   1:  PR[GP1:91,1] = PR[GP1:90,1] + -5.573;
   1:  PR[GP1:91,2] = PR[GP1:90,2] + 6.537;
   1:L PR[91] R[100]mm/sec CNT100;
   1:  PR[GP1:91,1] = PR[GP1:90,1] + -6.753;
   1:  PR[GP1:91,2] = PR[GP1:90,2] + 9.038;
   1:L PR[91] R[100]mm/sec CNT100;
   1:  PR[GP1:91,1] = PR[GP1:90,1] + -7.010;
   1:  PR[GP1:91,2] = PR[GP1:90,2] + 9.357;
   1:L PR[91] R[100]mm/sec CNT100;
   1:  PR[GP1:91,1] = PR[GP1:90,1] + -8.709;
   1:  PR[GP1:91,2] = PR[GP1:90,2] + 11.817;
   1:L PR[91] R[100]mm/sec CNT100;
   1:  PR[GP1:91,1] = PR[GP1:90,1] + -10.629;
   1:  PR[GP1:91,2] = PR[GP1:90,2] + 13.805;
   1:L PR[91] R[100]mm/sec CNT100;
   1:  PR[GP1:91,1] = PR[GP1:90,1] + -10.976;
   1:  PR[GP1:91,2] = PR[GP1:90,2] + 14.025;
   1:L PR[91] R[100]mm/sec CNT100;
   1:  PR[GP1:91,1] = PR[GP1:90,1] + -13.376;
   1:  PR[GP1:91,2] = PR[GP1:90,2] + 15.808;
   1:L PR[91] R[100]mm/sec CNT100;
   1:  PR[GP1:91,1] = PR[GP1:90,1] + -15.833;
   1:  PR[GP1:91,2] = PR[GP1:90,2] + 17.073;
   1:L PR[91] R[100]mm/sec CNT100;
   1:  PR[GP1:91,1] = PR[GP1:90,1] + -16.233;
   1:  PR[GP1:91,2] = PR[GP1:90,2] + 17.169;
   1:L PR[91] R[100]mm/sec CNT100;
   1:  PR[GP1:91,1] = PR[GP1:90,1] + -19.079;
   1:  PR[GP1:91,2] = PR[GP1:90,2] + 18.086;
   1:L PR[91] R[100]mm/sec CNT100;
   1:  PR[GP1:91,1] = PR[GP1:90,1] + -21.812;
   1:  PR[GP1:91,2] = PR[GP1:90,2] + 18.493;
   1:L PR[91] R[100]mm/sec CNT100;
   1:  PR[GP1:91,1] = PR[GP1:90,1] + -22.221;
   1:  PR[GP1:91,2] = PR[GP1:90,2] + 18.455;
   1:L PR[91] R[100]mm/sec CNT100;
   1:  PR[GP1:91,1] = PR[GP1:90,1] + -25.212;
   1:  PR[GP1:91,2] = PR[GP1:90,2] + 18.408;
   1:L PR[91] R[100]mm/sec CNT100;
   1:  PR[GP1:91,1] = PR[GP1:90,1] + -27.929;
   1:  PR[GP1:91,2] = PR[GP1:90,2] + 17.915;
   1:L PR[91] R[100]mm/sec CNT100;
   1:  PR[GP1:91,1] = PR[GP1:90,1] + -28.304;
   1:  PR[GP1:91,2] = PR[GP1:90,2] + 17.747;
   1:L PR[91] R[100]mm/sec CNT100;
   1:  PR[GP1:91,1] = PR[GP1:90,1] + -31.122;
   1:  PR[GP1:91,2] = PR[GP1:90,2] + 16.741;
   1:L PR[91] R[100]mm/sec CNT100;
   1:  PR[GP1:91,1] = PR[GP1:90,1] + -33.536;
   1:  PR[GP1:91,2] = PR[GP1:90,2] + 15.401;
   1:L PR[91] R[100]mm/sec CNT100;
   1:  PR[GP1:91,1] = PR[GP1:90,1] + -33.837;
   1:  PR[GP1:91,2] = PR[GP1:90,2] + 15.121;
   1:L PR[91] R[100]mm/sec CNT100;
   1:  PR[GP1:91,1] = PR[GP1:90,1] + -36.182;
   1:  PR[GP1:91,2] = PR[GP1:90,2] + 13.261;
   1:L PR[91] R[100]mm/sec CNT100;
   1:  PR[GP1:91,1] = PR[GP1:90,1] + -38.036;
   1:  PR[GP1:91,2] = PR[GP1:90,2] + 11.216;
   1:L PR[91] R[100]mm/sec CNT100;
   1:  PR[GP1:91,1] = PR[GP1:90,1] + -38.230;
   1:  PR[GP1:91,2] = PR[GP1:90,2] + 10.854;
   1:L PR[91] R[100]mm/sec CNT100;
   1:  PR[GP1:91,1] = PR[GP1:90,1] + -39.853;
   1:  PR[GP1:91,2] = PR[GP1:90,2] + 8.338;
   1:L PR[91] R[100]mm/sec CNT100;
   1:  PR[GP1:91,1] = PR[GP1:90,1] + -40.951;
   1:  PR[GP1:91,2] = PR[GP1:90,2] + 5.807;
   1:L PR[91] R[100]mm/sec CNT100;
   1:  PR[GP1:91,1] = PR[GP1:90,1] + -41.018;
   1:  PR[GP1:91,2] = PR[GP1:90,2] + 5.402;
   1:L PR[91] R[100]mm/sec CNT100;
   1:  PR[GP1:91,1] = PR[GP1:90,1] + -41.746;
   1:  PR[GP1:91,2] = PR[GP1:90,2] + 2.497;
   1:L PR[91] R[100]mm/sec CNT100;
   1:  PR[GP1:91,1] = PR[GP1:90,1] + -41.972;
   1:  PR[GP1:91,2] = PR[GP1:90,2] + -0.252;
   1:L PR[91] R[100]mm/sec CNT100;
   1:  PR[GP1:91,1] = PR[GP1:90,1] + -41.905;
   1:  PR[GP1:91,2] = PR[GP1:90,2] + -0.657;
   1:L PR[91] R[100]mm/sec CNT100;
   1:  PR[GP1:91,1] = PR[GP1:90,1] + -41.660;
   1:  PR[GP1:91,2] = PR[GP1:90,2] + -3.643;
   1:L PR[91] R[100]mm/sec CNT100;
   1:  PR[GP1:91,1] = PR[GP1:90,1] + -40.975;
   1:  PR[GP1:91,2] = PR[GP1:90,2] + -6.377;
   1:L PR[91] R[100]mm/sec CNT100;
   1:  PR[GP1:91,1] = PR[GP1:90,1] + -39.830;
   1:  PR[GP1:91,2] = PR[GP1:90,2] + -9.016;
   1:L PR[91] R[100]mm/sec CNT100;
   1:  PR[GP1:91,1] = PR[GP1:90,1] + -39.636;
   1:  PR[GP1:91,2] = PR[GP1:90,2] + -9.378;
   1:L PR[91] R[100]mm/sec CNT100;
   1:  PR[GP1:91,1] = PR[GP1:90,1] + -38.075;
   1:  PR[GP1:91,2] = PR[GP1:90,2] + -11.797;
   1:L PR[91] R[100]mm/sec CNT100;
   1:  PR[GP1:91,1] = PR[GP1:90,1] + -36.144;
   1:  PR[GP1:91,2] = PR[GP1:90,2] + -13.927;
   1:L PR[91] R[100]mm/sec CNT100;
   1:  PR[GP1:91,1] = PR[GP1:90,1] + -35.842;
   1:  PR[GP1:91,2] = PR[GP1:90,2] + -14.207;
   1:L PR[91] R[100]mm/sec CNT100;
   1:  PR[GP1:91,1] = PR[GP1:90,1] + -33.586;
   1:  PR[GP1:91,2] = PR[GP1:90,2] + -15.997;
   1:L PR[91] R[100]mm/sec CNT100;
   1:  PR[GP1:91,1] = PR[GP1:90,1] + -31.073;
   1:  PR[GP1:91,2] = PR[GP1:90,2] + -17.392;
   1:L PR[91] R[100]mm/sec CNT100;
   1:  PR[GP1:91,1] = PR[GP1:90,1] + -30.697;
   1:  PR[GP1:91,2] = PR[GP1:90,2] + -17.560;
   1:L PR[91] R[100]mm/sec CNT100;
   1:  PR[GP1:91,1] = PR[GP1:90,1] + -27.985;
   1:  PR[GP1:91,2] = PR[GP1:90,2] + -18.529;
   1:L PR[91] R[100]mm/sec CNT100;
   1:  PR[GP1:91,1] = PR[GP1:90,1] + -25.157;
   1:  PR[GP1:91,2] = PR[GP1:90,2] + -19.042;
   1:L PR[91] R[100]mm/sec CNT100;
   1:  PR[GP1:91,1] = PR[GP1:90,1] + -24.748;
   1:  PR[GP1:91,2] = PR[GP1:90,2] + -19.080;
   1:L PR[91] R[100]mm/sec CNT100;
   1:  PR[GP1:91,1] = PR[GP1:90,1] + -21.867;
   1:  PR[GP1:91,2] = PR[GP1:90,2] + -19.125;
   1:L PR[91] R[100]mm/sec CNT100;
   1:  PR[GP1:91,1] = PR[GP1:90,1] + -19.025;
   1:  PR[GP1:91,2] = PR[GP1:90,2] + -18.702;
   1:L PR[91] R[100]mm/sec CNT100;
   1:  PR[GP1:91,1] = PR[GP1:90,1] + -18.625;
   1:  PR[GP1:91,2] = PR[GP1:90,2] + -18.606;
   1:L PR[91] R[100]mm/sec CNT100;
   1:  PR[GP1:91,1] = PR[GP1:90,1] + -15.882;
   1:  PR[GP1:91,2] = PR[GP1:90,2] + -17.722;
   1:L PR[91] R[100]mm/sec CNT100;
   1:  PR[GP1:91,1] = PR[GP1:90,1] + -13.329;
   1:  PR[GP1:91,2] = PR[GP1:90,2] + -16.408;
   1:L PR[91] R[100]mm/sec CNT100;
   1:  PR[GP1:91,1] = PR[GP1:90,1] + -12.981;
   1:  PR[GP1:91,2] = PR[GP1:90,2] + -16.187;
   1:L PR[91] R[100]mm/sec CNT100;
   1:  PR[GP1:91,1] = PR[GP1:90,1] + -10.667;
   1:  PR[GP1:91,2] = PR[GP1:90,2] + -14.468;
   1:L PR[91] R[100]mm/sec CNT100;
   1:  PR[GP1:91,1] = PR[GP1:90,1] + -8.672;
   1:  PR[GP1:91,2] = PR[GP1:90,2] + -12.403;
   1:L PR[91] R[100]mm/sec CNT100;
   1:  PR[GP1:91,1] = PR[GP1:90,1] + -8.414;
   1:  PR[GP1:91,2] = PR[GP1:90,2] + -12.082;
   1:L PR[91] R[100]mm/sec CNT100;
   1:  PR[GP1:91,1] = PR[GP1:90,1] + -6.775;
   1:  PR[GP1:91,2] = PR[GP1:90,2] + -9.710;
   1:L PR[91] R[100]mm/sec CNT100;
   1:  PR[GP1:91,1] = PR[GP1:90,1] + -5.551;
   1:  PR[GP1:91,2] = PR[GP1:90,2] + -7.113;
   1:L PR[91] R[100]mm/sec CNT100;
   1:  PR[GP1:91,1] = PR[GP1:90,1] + -5.411;
   1:  PR[GP1:91,2] = PR[GP1:90,2] + -6.729;
   1:L PR[91] R[100]mm/sec CNT100;
   1:  PR[GP1:91,1] = PR[GP1:90,1] + -4.557;
   1:  PR[GP1:91,2] = PR[GP1:90,2] + -3.704;
   1:L PR[91] R[100]mm/sec CNT100;
   1:  PR[GP1:91,1] = PR[GP1:90,1] + -4.234;
   1:  PR[GP1:91,2] = PR[GP1:90,2] + -2.880;
   1:L PR[91] R[100]mm/sec CNT100;
   1:  PR[GP1:91,1] = PR[GP1:90,1] + -3.519;
   1:  PR[GP1:91,2] = PR[GP1:90,2] + -2.050;
   1:L PR[91] R[100]mm/sec CNT100;
   1:  PR[GP1:91,1] = PR[GP1:90,1] + -2.563;
   1:  PR[GP1:91,2] = PR[GP1:90,2] + -1.510;
   1:L PR[91] R[100]mm/sec CNT100;
   1:  PR[GP1:91,1] = PR[GP1:90,1] + -2.182;
   1:  PR[GP1:91,2] = PR[GP1:90,2] + -1.443;
   1:L PR[91] R[100]mm/sec CNT100;
   1:  PR[GP1:91,1] = PR[GP1:90,1] + -1.745;
   1:  PR[GP1:91,2] = PR[GP1:90,2] + -1.269;
   1:L PR[91] R[100]mm/sec CNT100;
   1:  PR[GP1:91,1] = PR[GP1:90,1] + 1.895;
   1:  PR[GP1:91,2] = PR[GP1:90,2] + -1.275;
   1:L PR[91] R[100]mm/sec CNT100;
   1:  PR[GP1:91,1] = PR[GP1:90,1] + 2.330;
   1:  PR[GP1:91,2] = PR[GP1:90,2] + -1.442;
   1:L PR[91] R[100]mm/sec CNT100;
   1:  PR[GP1:91,1] = PR[GP1:90,1] + 2.720;
   1:  PR[GP1:91,2] = PR[GP1:90,2] + -1.510;
   1:L PR[91] R[100]mm/sec CNT100;
   1:  PR[GP1:91,1] = PR[GP1:90,1] + 3.676;
   1:  PR[GP1:91,2] = PR[GP1:90,2] + -2.050;
   1:L PR[91] R[100]mm/sec CNT100;
   1:  PR[GP1:91,1] = PR[GP1:90,1] + 4.391;
   1:  PR[GP1:91,2] = PR[GP1:90,2] + -2.881;
   1:L PR[91] R[100]mm/sec CNT100;
   1:  PR[GP1:91,1] = PR[GP1:90,1] + 4.700;
   1:  PR[GP1:91,2] = PR[GP1:90,2] + -3.670;
   1:L PR[91] R[100]mm/sec CNT100;
   1:  PR[GP1:91,1] = PR[GP1:90,1] + 4.916;
   1:  PR[GP1:91,2] = PR[GP1:90,2] + -4.299;
   1:L PR[91] R[100]mm/sec CNT100;
   1:  PR[GP1:91,1] = PR[GP1:90,1] + 5.730;
   1:  PR[GP1:91,2] = PR[GP1:90,2] + -7.161;
   1:L PR[91] R[100]mm/sec CNT100;
   1:  PR[GP1:91,1] = PR[GP1:90,1] + 6.909;
   1:  PR[GP1:91,2] = PR[GP1:90,2] + -9.661;
   1:L PR[91] R[100]mm/sec CNT100;
   1:  PR[GP1:91,1] = PR[GP1:90,1] + 7.167;
   1:  PR[GP1:91,2] = PR[GP1:90,2] + -9.981;
   1:L PR[91] R[100]mm/sec CNT100;
   1:  PR[GP1:91,1] = PR[GP1:90,1] + 8.866;
   1:  PR[GP1:91,2] = PR[GP1:90,2] + -12.441;
   1:L PR[91] R[100]mm/sec CNT100;
   1:  PR[GP1:91,1] = PR[GP1:90,1] + 10.786;
   1:  PR[GP1:91,2] = PR[GP1:90,2] + -14.429;
   1:L PR[91] R[100]mm/sec CNT100;
   1:  PR[GP1:91,1] = PR[GP1:90,1] + 11.133;
   1:  PR[GP1:91,2] = PR[GP1:90,2] + -14.649;
   1:L PR[91] R[100]mm/sec CNT100;
   1:  PR[GP1:91,1] = PR[GP1:90,1] + 13.533;
   1:  PR[GP1:91,2] = PR[GP1:90,2] + -16.432;
   1:L PR[91] R[100]mm/sec CNT100;
   1:  PR[GP1:91,1] = PR[GP1:90,1] + 15.990;
   1:  PR[GP1:91,2] = PR[GP1:90,2] + -17.697;
   1:L PR[91] R[100]mm/sec CNT100;
   1:  PR[GP1:91,1] = PR[GP1:90,1] + 16.389;
   1:  PR[GP1:91,2] = PR[GP1:90,2] + -17.793;
   1:L PR[91] R[100]mm/sec CNT100;
   1:  PR[GP1:91,1] = PR[GP1:90,1] + 19.236;
   1:  PR[GP1:91,2] = PR[GP1:90,2] + -18.710;
   1:L PR[91] R[100]mm/sec CNT100;
   1:  PR[GP1:91,1] = PR[GP1:90,1] + 21.968;
   1:  PR[GP1:91,2] = PR[GP1:90,2] + -19.117;
   1:L PR[91] R[100]mm/sec CNT100;
   1:  PR[GP1:91,1] = PR[GP1:90,1] + 22.377;
   1:  PR[GP1:91,2] = PR[GP1:90,2] + -19.079;
   1:L PR[91] R[100]mm/sec CNT100;
   1:  PR[GP1:91,1] = PR[GP1:90,1] + 25.369;
   1:  PR[GP1:91,2] = PR[GP1:90,2] + -19.032;
   1:L PR[91] R[100]mm/sec CNT100;
   1:  PR[GP1:91,1] = PR[GP1:90,1] + 28.086;
   1:  PR[GP1:91,2] = PR[GP1:90,2] + -18.539;
   1:L PR[91] R[100]mm/sec CNT100;
   1:  PR[GP1:91,1] = PR[GP1:90,1] + 28.461;
   1:  PR[GP1:91,2] = PR[GP1:90,2] + -18.371;
   1:L PR[91] R[100]mm/sec CNT100;
   1:  PR[GP1:91,1] = PR[GP1:90,1] + 31.279;
   1:  PR[GP1:91,2] = PR[GP1:90,2] + -17.365;
   1:L PR[91] R[100]mm/sec CNT100;
   1:  PR[GP1:91,1] = PR[GP1:90,1] + 33.693;
   1:  PR[GP1:91,2] = PR[GP1:90,2] + -16.025;
   1:L PR[91] R[100]mm/sec CNT100;
   1:  PR[GP1:91,1] = PR[GP1:90,1] + 33.993;
   1:  PR[GP1:91,2] = PR[GP1:90,2] + -15.745;
   1:L PR[91] R[100]mm/sec CNT100;
   1:  PR[GP1:91,1] = PR[GP1:90,1] + 36.339;
   1:  PR[GP1:91,2] = PR[GP1:90,2] + -13.885;
   1:L PR[91] R[100]mm/sec CNT100;
   1:  PR[GP1:91,1] = PR[GP1:90,1] + 38.193;
   1:  PR[GP1:91,2] = PR[GP1:90,2] + -11.840;
   1:L PR[91] R[100]mm/sec CNT100;
   1:  PR[GP1:91,1] = PR[GP1:90,1] + 38.387;
   1:  PR[GP1:91,2] = PR[GP1:90,2] + -11.478;
   1:L PR[91] R[100]mm/sec CNT100;
   1:  PR[GP1:91,1] = PR[GP1:90,1] + 40.010;
   1:  PR[GP1:91,2] = PR[GP1:90,2] + -8.962;
   1:L PR[91] R[100]mm/sec CNT100;
   1:  PR[GP1:91,1] = PR[GP1:90,1] + 41.108;
   1:  PR[GP1:91,2] = PR[GP1:90,2] + -6.431;
   1:L PR[91] R[100]mm/sec CNT100;
   1:  PR[GP1:91,1] = PR[GP1:90,1] + 41.175;
   1:  PR[GP1:91,2] = PR[GP1:90,2] + -6.026;
   1:L PR[91] R[100]mm/sec CNT100;
   1:  PR[GP1:91,1] = PR[GP1:90,1] + 41.903;
   1:  PR[GP1:91,2] = PR[GP1:90,2] + -3.121;
   1:L PR[91] R[100]mm/sec CNT100;
   1:  PR[GP1:91,1] = PR[GP1:90,1] + 42.129;
   1:  PR[GP1:91,2] = PR[GP1:90,2] + -0.372;
   1:L PR[91] R[100]mm/sec CNT100;
   1:  PR[GP1:91,1] = PR[GP1:90,1] + 42.061;
   1:  PR[GP1:91,2] = PR[GP1:90,2] + 0.033;
   1:L PR[91] R[100]mm/sec CNT100;
   1:  PR[GP1:91,1] = PR[GP1:90,1] + 41.817;
   1:  PR[GP1:91,2] = PR[GP1:90,2] + 3.019;
   1:L PR[91] R[100]mm/sec CNT100;
   1:  PR[GP1:91,1] = PR[GP1:90,1] + 41.132;
   1:  PR[GP1:91,2] = PR[GP1:90,2] + 5.753;
   1:L PR[91] R[100]mm/sec CNT100;
   1:  PR[GP1:91,1] = PR[GP1:90,1] + 39.987;
   1:  PR[GP1:91,2] = PR[GP1:90,2] + 8.392;
   1:L PR[91] R[100]mm/sec CNT100;
   1:  PR[GP1:91,1] = PR[GP1:90,1] + 39.792;
   1:  PR[GP1:91,2] = PR[GP1:90,2] + 8.754;
   1:L PR[91] R[100]mm/sec CNT100;
   1:  PR[GP1:91,1] = PR[GP1:90,1] + 38.232;
   1:  PR[GP1:91,2] = PR[GP1:90,2] + 11.173;
   1:L PR[91] R[100]mm/sec CNT100;
   1:  PR[GP1:91,1] = PR[GP1:90,1] + 36.300;
   1:  PR[GP1:91,2] = PR[GP1:90,2] + 13.303;
   1:L PR[91] R[100]mm/sec CNT100;
   1:  PR[GP1:91,1] = PR[GP1:90,1] + 35.999;
   1:  PR[GP1:91,2] = PR[GP1:90,2] + 13.583;
   1:L PR[91] R[100]mm/sec CNT100;
   1:  PR[GP1:91,1] = PR[GP1:90,1] + 33.743;
   1:  PR[GP1:91,2] = PR[GP1:90,2] + 15.373;
   1:L PR[91] R[100]mm/sec CNT100;
   1:  PR[GP1:91,1] = PR[GP1:90,1] + 31.230;
   1:  PR[GP1:91,2] = PR[GP1:90,2] + 16.768;
   1:L PR[91] R[100]mm/sec CNT100;
   1:  PR[GP1:91,1] = PR[GP1:90,1] + 30.854;
   1:  PR[GP1:91,2] = PR[GP1:90,2] + 16.936;
   1:L PR[91] R[100]mm/sec CNT100;
   1:  PR[GP1:91,1] = PR[GP1:90,1] + 28.142;
   1:  PR[GP1:91,2] = PR[GP1:90,2] + 17.905;
   1:L PR[91] R[100]mm/sec CNT100;
   1:  PR[GP1:91,1] = PR[GP1:90,1] + 25.314;
   1:  PR[GP1:91,2] = PR[GP1:90,2] + 18.418;
   1:L PR[91] R[100]mm/sec CNT100;
   1:  PR[GP1:91,1] = PR[GP1:90,1] + 24.904;
   1:  PR[GP1:91,2] = PR[GP1:90,2] + 18.456;
   1:L PR[91] R[100]mm/sec CNT100;
   1:  PR[GP1:91,1] = PR[GP1:90,1] + 22.024;
   1:  PR[GP1:91,2] = PR[GP1:90,2] + 18.501;
   1:L PR[91] R[100]mm/sec CNT100;
   1:  PR[GP1:91,1] = PR[GP1:90,1] + 19.182;
   1:  PR[GP1:91,2] = PR[GP1:90,2] + 18.078;
   1:L PR[91] R[100]mm/sec CNT100;
   1:  PR[GP1:91,1] = PR[GP1:90,1] + 18.782;
   1:  PR[GP1:91,2] = PR[GP1:90,2] + 17.982;
   1:L PR[91] R[100]mm/sec CNT100;
   1:  PR[GP1:91,1] = PR[GP1:90,1] + 16.039;
   1:  PR[GP1:91,2] = PR[GP1:90,2] + 17.098;
   1:L PR[91] R[100]mm/sec CNT100;
   1:  PR[GP1:91,1] = PR[GP1:90,1] + 13.485;
   1:  PR[GP1:91,2] = PR[GP1:90,2] + 15.784;
   1:L PR[91] R[100]mm/sec CNT100;
   1:  PR[GP1:91,1] = PR[GP1:90,1] + 13.138;
   1:  PR[GP1:91,2] = PR[GP1:90,2] + 15.563;
   1:L PR[91] R[100]mm/sec CNT100;
   1:  PR[GP1:91,1] = PR[GP1:90,1] + 10.824;
   1:  PR[GP1:91,2] = PR[GP1:90,2] + 13.844;
   1:L PR[91] R[100]mm/sec CNT100;
   1:  PR[GP1:91,1] = PR[GP1:90,1] + 8.829;
   1:  PR[GP1:91,2] = PR[GP1:90,2] + 11.779;
   1:L PR[91] R[100]mm/sec CNT100;
   1:  PR[GP1:91,1] = PR[GP1:90,1] + 8.571;
   1:  PR[GP1:91,2] = PR[GP1:90,2] + 11.459;
   1:L PR[91] R[100]mm/sec CNT100;
   1:  PR[GP1:91,1] = PR[GP1:90,1] + 6.932;
   1:  PR[GP1:91,2] = PR[GP1:90,2] + 9.086;
   1:L PR[91] R[100]mm/sec CNT100;
   1:  PR[GP1:91,1] = PR[GP1:90,1] + 5.708;
   1:  PR[GP1:91,2] = PR[GP1:90,2] + 6.489;
   1:L PR[91] R[100]mm/sec CNT100;
   1:  PR[GP1:91,1] = PR[GP1:90,1] + 5.568;
   1:  PR[GP1:91,2] = PR[GP1:90,2] + 6.105;
   1:L PR[91] R[100]mm/sec CNT100;
   1:  PR[GP1:91,1] = PR[GP1:90,1] + 4.714;
   1:  PR[GP1:91,2] = PR[GP1:90,2] + 3.080;
   1:L PR[91] R[100]mm/sec CNT100;
   1:  PR[GP1:91,1] = PR[GP1:90,1] + 4.391;
   1:  PR[GP1:91,2] = PR[GP1:90,2] + 2.256;
   1:L PR[91] R[100]mm/sec CNT100;
   1:  PR[GP1:91,1] = PR[GP1:90,1] + 3.676;
   1:  PR[GP1:91,2] = PR[GP1:90,2] + 1.426;
   1:L PR[91] R[100]mm/sec CNT100;
   1:  PR[GP1:91,1] = PR[GP1:90,1] + 2.720;
   1:  PR[GP1:91,2] = PR[GP1:90,2] + 0.886;
   1:L PR[91] R[100]mm/sec CNT100;
   1:  PR[GP1:91,1] = PR[GP1:90,1] + 2.341;
   1:  PR[GP1:91,2] = PR[GP1:90,2] + 0.820;
   1:L PR[91] R[100]mm/sec CNT100;
   1:  PR[GP1:91,1] = PR[GP1:90,1] + 1.903;
   1:  PR[GP1:91,2] = PR[GP1:90,2] + 0.644;
   1:L PR[91] R[100]mm/sec CNT100;
   1:  PR[GP1:91,1] = PR[GP1:90,1] + -1.738;
   1:  PR[GP1:91,2] = PR[GP1:90,2] + 0.651;
   1:L PR[91] R[100]mm/sec CNT100;
   1:  PR[91] = PR[90];
   1:  PR[GP1:91,1] = PR[GP1:90,1] + -2.253;
   1:  PR[GP1:91,2] = PR[GP1:90,2] + 0.908;
   1:  PR[GP1:91,3] = PR[GP1:90,3] + 5.185;
   1:L PR[91] R[100]mm/sec CNT100;
   1:  PR[GP1:91,1] = PR[GP1:90,1] + -2.647;
   1:  PR[GP1:91,2] = PR[GP1:90,2] + 1.025;
   1:L PR[91] R[100]mm/sec CNT100;
   1:  PR[GP1:91,1] = PR[GP1:90,1] + -3.536;
   1:  PR[GP1:91,2] = PR[GP1:90,2] + 1.523;
   1:L PR[91] R[100]mm/sec CNT100;
   1:  PR[GP1:91,1] = PR[GP1:90,1] + -4.259;
   1:  PR[GP1:91,2] = PR[GP1:90,2] + 2.372;
   1:L PR[91] R[100]mm/sec CNT100;
   1:  PR[GP1:91,1] = PR[GP1:90,1] + -4.588;
   1:  PR[GP1:91,2] = PR[GP1:90,2] + 3.246;
   1:L PR[91] R[100]mm/sec CNT100;
   1:  PR[GP1:91,1] = PR[GP1:90,1] + -5.418;
   1:  PR[GP1:91,2] = PR[GP1:90,2] + 6.210;
   1:L PR[91] R[100]mm/sec CNT100;
   1:  PR[GP1:91,1] = PR[GP1:90,1] + -6.705;
   1:  PR[GP1:91,2] = PR[GP1:90,2] + 8.939;
   1:L PR[91] R[100]mm/sec CNT100;
   1:  PR[GP1:91,1] = PR[GP1:90,1] + -6.791;
   1:  PR[GP1:91,2] = PR[GP1:90,2] + 9.139;
   1:L PR[91] R[100]mm/sec CNT100;
   1:  PR[GP1:91,1] = PR[GP1:90,1] + -8.462;
   1:  PR[GP1:91,2] = PR[GP1:90,2] + 11.559;
   1:L PR[91] R[100]mm/sec CNT100;
   1:  PR[GP1:91,1] = PR[GP1:90,1] + -8.569;
   1:  PR[GP1:91,2] = PR[GP1:90,2] + 11.694;
   1:L PR[91] R[100]mm/sec CNT100;
   1:  PR[GP1:91,1] = PR[GP1:90,1] + -10.621;
   1:  PR[GP1:91,2] = PR[GP1:90,2] + 13.818;
   1:L PR[91] R[100]mm/sec CNT100;
   1:  PR[GP1:91,1] = PR[GP1:90,1] + -13.178;
   1:  PR[GP1:91,2] = PR[GP1:90,2] + 15.718;
   1:L PR[91] R[100]mm/sec CNT100;
   1:  PR[GP1:91,1] = PR[GP1:90,1] + -15.815;
   1:  PR[GP1:91,2] = PR[GP1:90,2] + 17.075;
   1:L PR[91] R[100]mm/sec CNT100;
   1:  PR[GP1:91,1] = PR[GP1:90,1] + -15.944;
   1:  PR[GP1:91,2] = PR[GP1:90,2] + 17.127;
   1:L PR[91] R[100]mm/sec CNT100;
   1:  PR[GP1:91,1] = PR[GP1:90,1] + -18.795;
   1:  PR[GP1:91,2] = PR[GP1:90,2] + 18.045;
   1:L PR[91] R[100]mm/sec CNT100;
   1:  PR[GP1:91,1] = PR[GP1:90,1] + -21.788;
   1:  PR[GP1:91,2] = PR[GP1:90,2] + 18.491;
   1:L PR[91] R[100]mm/sec CNT100;
   1:  PR[GP1:91,1] = PR[GP1:90,1] + -21.912;
   1:  PR[GP1:91,2] = PR[GP1:90,2] + 18.506;
   1:L PR[91] R[100]mm/sec CNT100;
   1:  PR[GP1:91,1] = PR[GP1:90,1] + -24.871;
   1:  PR[GP1:91,2] = PR[GP1:90,2] + 18.460;
   1:L PR[91] R[100]mm/sec CNT100;
   1:  PR[GP1:91,1] = PR[GP1:90,1] + -27.991;
   1:  PR[GP1:91,2] = PR[GP1:90,2] + 17.902;
   1:L PR[91] R[100]mm/sec CNT100;
   1:  PR[GP1:91,1] = PR[GP1:90,1] + -30.837;
   1:  PR[GP1:91,2] = PR[GP1:90,2] + 16.886;
   1:L PR[91] R[100]mm/sec CNT100;
   1:  PR[GP1:91,1] = PR[GP1:90,1] + -30.925;
   1:  PR[GP1:91,2] = PR[GP1:90,2] + 16.849;
   1:L PR[91] R[100]mm/sec CNT100;
   1:  PR[GP1:91,1] = PR[GP1:90,1] + -33.543;
   1:  PR[GP1:91,2] = PR[GP1:90,2] + 15.395;
   1:L PR[91] R[100]mm/sec CNT100;
   1:  PR[GP1:91,1] = PR[GP1:90,1] + -36.018;
   1:  PR[GP1:91,2] = PR[GP1:90,2] + 13.434;
   1:L PR[91] R[100]mm/sec CNT100;
   1:  PR[GP1:91,1] = PR[GP1:90,1] + -38.044;
   1:  PR[GP1:91,2] = PR[GP1:90,2] + 11.201;
   1:L PR[91] R[100]mm/sec CNT100;
   1:  PR[GP1:91,1] = PR[GP1:90,1] + -38.090;
   1:  PR[GP1:91,2] = PR[GP1:90,2] + 11.140;
   1:L PR[91] R[100]mm/sec CNT100;
   1:  PR[GP1:91,1] = PR[GP1:90,1] + -39.729;
   1:  PR[GP1:91,2] = PR[GP1:90,2] + 8.599;
   1:L PR[91] R[100]mm/sec CNT100;
   1:  PR[GP1:91,1] = PR[GP1:90,1] + -40.981;
   1:  PR[GP1:91,2] = PR[GP1:90,2] + 5.706;
   1:L PR[91] R[100]mm/sec CNT100;
   1:  PR[GP1:91,1] = PR[GP1:90,1] + -41.702;
   1:  PR[GP1:91,2] = PR[GP1:90,2] + 2.827;
   1:L PR[91] R[100]mm/sec CNT100;
   1:  PR[GP1:91,1] = PR[GP1:90,1] + -41.968;
   1:  PR[GP1:91,2] = PR[GP1:90,2] + -0.312;
   1:L PR[91] R[100]mm/sec CNT100;
   1:  PR[GP1:91,1] = PR[GP1:90,1] + -41.702;
   1:  PR[GP1:91,2] = PR[GP1:90,2] + -3.451;
   1:L PR[91] R[100]mm/sec CNT100;
   1:  PR[GP1:91,1] = PR[GP1:90,1] + -40.981;
   1:  PR[GP1:91,2] = PR[GP1:90,2] + -6.330;
   1:L PR[91] R[100]mm/sec CNT100;
   1:  PR[GP1:91,1] = PR[GP1:90,1] + -39.729;
   1:  PR[GP1:91,2] = PR[GP1:90,2] + -9.223;
   1:L PR[91] R[100]mm/sec CNT100;
   1:  PR[GP1:91,1] = PR[GP1:90,1] + -38.090;
   1:  PR[GP1:91,2] = PR[GP1:90,2] + -11.764;
   1:L PR[91] R[100]mm/sec CNT100;
   1:  PR[GP1:91,1] = PR[GP1:90,1] + -38.044;
   1:  PR[GP1:91,2] = PR[GP1:90,2] + -11.825;
   1:L PR[91] R[100]mm/sec CNT100;
   1:  PR[GP1:91,1] = PR[GP1:90,1] + -36.018;
   1:  PR[GP1:91,2] = PR[GP1:90,2] + -14.058;
   1:L PR[91] R[100]mm/sec CNT100;
   1:  PR[GP1:91,1] = PR[GP1:90,1] + -33.543;
   1:  PR[GP1:91,2] = PR[GP1:90,2] + -16.019;
   1:L PR[91] R[100]mm/sec CNT100;
   1:  PR[GP1:91,1] = PR[GP1:90,1] + -30.925;
   1:  PR[GP1:91,2] = PR[GP1:90,2] + -17.473;
   1:L PR[91] R[100]mm/sec CNT100;
   1:  PR[GP1:91,1] = PR[GP1:90,1] + -30.837;
   1:  PR[GP1:91,2] = PR[GP1:90,2] + -17.509;
   1:L PR[91] R[100]mm/sec CNT100;
   1:  PR[GP1:91,1] = PR[GP1:90,1] + -27.991;
   1:  PR[GP1:91,2] = PR[GP1:90,2] + -18.526;
   1:L PR[91] R[100]mm/sec CNT100;
   1:  PR[GP1:91,1] = PR[GP1:90,1] + -24.871;
   1:  PR[GP1:91,2] = PR[GP1:90,2] + -19.084;
   1:L PR[91] R[100]mm/sec CNT100;
   1:  PR[GP1:91,1] = PR[GP1:90,1] + -21.931;
   1:  PR[GP1:91,2] = PR[GP1:90,2] + -19.130;
   1:L PR[91] R[100]mm/sec CNT100;
   1:  PR[GP1:91,1] = PR[GP1:90,1] + -18.794;
   1:  PR[GP1:91,2] = PR[GP1:90,2] + -18.669;
   1:L PR[91] R[100]mm/sec CNT100;
   1:  PR[GP1:91,1] = PR[GP1:90,1] + -15.944;
   1:  PR[GP1:91,2] = PR[GP1:90,2] + -17.751;
   1:L PR[91] R[100]mm/sec CNT100;
   1:  PR[GP1:91,1] = PR[GP1:90,1] + -15.815;
   1:  PR[GP1:91,2] = PR[GP1:90,2] + -17.699;
   1:L PR[91] R[100]mm/sec CNT100;
   1:  PR[GP1:91,1] = PR[GP1:90,1] + -13.178;
   1:  PR[GP1:91,2] = PR[GP1:90,2] + -16.342;
   1:L PR[91] R[100]mm/sec CNT100;
   1:  PR[GP1:91,1] = PR[GP1:90,1] + -10.621;
   1:  PR[GP1:91,2] = PR[GP1:90,2] + -14.442;
   1:L PR[91] R[100]mm/sec CNT100;
   1:  PR[GP1:91,1] = PR[GP1:90,1] + -8.569;
   1:  PR[GP1:91,2] = PR[GP1:90,2] + -12.318;
   1:L PR[91] R[100]mm/sec CNT100;
   1:  PR[GP1:91,1] = PR[GP1:90,1] + -8.462;
   1:  PR[GP1:91,2] = PR[GP1:90,2] + -12.183;
   1:L PR[91] R[100]mm/sec CNT100;
   1:  PR[GP1:91,1] = PR[GP1:90,1] + -6.777;
   1:  PR[GP1:91,2] = PR[GP1:90,2] + -9.743;
   1:L PR[91] R[100]mm/sec CNT100;
   1:  PR[GP1:91,1] = PR[GP1:90,1] + -5.421;
   1:  PR[GP1:91,2] = PR[GP1:90,2] + -6.847;
   1:L PR[91] R[100]mm/sec CNT100;
   1:  PR[GP1:91,1] = PR[GP1:90,1] + -4.741;
   1:  PR[GP1:91,2] = PR[GP1:90,2] + -4.458;
   1:L PR[91] R[100]mm/sec CNT100;
   1:  PR[GP1:91,1] = PR[GP1:90,1] + -4.779;
   1:  PR[GP1:91,2] = PR[GP1:90,2] + -4.375;
   1:L PR[91] R[100]mm/sec CNT100;
   1:  PR[GP1:91,1] = PR[GP1:90,1] + -4.259;
   1:  PR[GP1:91,2] = PR[GP1:90,2] + -2.996;
   1:L PR[91] R[100]mm/sec CNT100;
   1:  PR[GP1:91,1] = PR[GP1:90,1] + -3.536;
   1:  PR[GP1:91,2] = PR[GP1:90,2] + -2.147;
   1:L PR[91] R[100]mm/sec CNT100;
   1:  PR[GP1:91,1] = PR[GP1:90,1] + -2.648;
   1:  PR[GP1:91,2] = PR[GP1:90,2] + -1.649;
   1:L PR[91] R[100]mm/sec CNT100;
   1:  PR[GP1:91,1] = PR[GP1:90,1] + -2.234;
   1:  PR[GP1:91,2] = PR[GP1:90,2] + -1.527;
   1:L PR[91] R[100]mm/sec CNT100;
   1:  PR[GP1:91,1] = PR[GP1:90,1] + -1.613;
   1:  PR[GP1:91,2] = PR[GP1:90,2] + -1.419;
   1:L PR[91] R[100]mm/sec CNT100;
   1:  PR[GP1:91,1] = PR[GP1:90,1] + 1.771;
   1:  PR[GP1:91,2] = PR[GP1:90,2] + -1.422;
   1:L PR[91] R[100]mm/sec CNT100;
   1:  PR[GP1:91,1] = PR[GP1:90,1] + 2.409;
   1:  PR[GP1:91,2] = PR[GP1:90,2] + -1.532;
   1:L PR[91] R[100]mm/sec CNT100;
   1:  PR[GP1:91,1] = PR[GP1:90,1] + 2.804;
   1:  PR[GP1:91,2] = PR[GP1:90,2] + -1.649;
   1:L PR[91] R[100]mm/sec CNT100;
   1:  PR[GP1:91,1] = PR[GP1:90,1] + 3.692;
   1:  PR[GP1:91,2] = PR[GP1:90,2] + -2.147;
   1:L PR[91] R[100]mm/sec CNT100;
   1:  PR[GP1:91,1] = PR[GP1:90,1] + 4.415;
   1:  PR[GP1:91,2] = PR[GP1:90,2] + -2.996;
   1:L PR[91] R[100]mm/sec CNT100;
   1:  PR[GP1:91,1] = PR[GP1:90,1] + 4.745;
   1:  PR[GP1:91,2] = PR[GP1:90,2] + -3.871;
   1:L PR[91] R[100]mm/sec CNT100;
   1:  PR[GP1:91,1] = PR[GP1:90,1] + 5.576;
   1:  PR[GP1:91,2] = PR[GP1:90,2] + -6.837;
   1:L PR[91] R[100]mm/sec CNT100;
   1:  PR[GP1:91,1] = PR[GP1:90,1] + 6.864;
   1:  PR[GP1:91,2] = PR[GP1:90,2] + -9.568;
   1:L PR[91] R[100]mm/sec CNT100;
   1:  PR[GP1:91,1] = PR[GP1:90,1] + 6.947;
   1:  PR[GP1:91,2] = PR[GP1:90,2] + -9.762;
   1:L PR[91] R[100]mm/sec CNT100;
   1:  PR[GP1:91,1] = PR[GP1:90,1] + 8.619;
   1:  PR[GP1:91,2] = PR[GP1:90,2] + -12.183;
   1:L PR[91] R[100]mm/sec CNT100;
   1:  PR[GP1:91,1] = PR[GP1:90,1] + 8.726;
   1:  PR[GP1:91,2] = PR[GP1:90,2] + -12.318;
   1:L PR[91] R[100]mm/sec CNT100;
   1:  PR[GP1:91,1] = PR[GP1:90,1] + 10.778;
   1:  PR[GP1:91,2] = PR[GP1:90,2] + -14.442;
   1:L PR[91] R[100]mm/sec CNT100;
   1:  PR[GP1:91,1] = PR[GP1:90,1] + 13.335;
   1:  PR[GP1:91,2] = PR[GP1:90,2] + -16.342;
   1:L PR[91] R[100]mm/sec CNT100;
   1:  PR[GP1:91,1] = PR[GP1:90,1] + 15.972;
   1:  PR[GP1:91,2] = PR[GP1:90,2] + -17.699;
   1:L PR[91] R[100]mm/sec CNT100;
   1:  PR[GP1:91,1] = PR[GP1:90,1] + 16.100;
   1:  PR[GP1:91,2] = PR[GP1:90,2] + -17.751;
   1:L PR[91] R[100]mm/sec CNT100;
   1:  PR[GP1:91,1] = PR[GP1:90,1] + 18.952;
   1:  PR[GP1:91,2] = PR[GP1:90,2] + -18.669;
   1:L PR[91] R[100]mm/sec CNT100;
   1:  PR[GP1:91,1] = PR[GP1:90,1] + 21.945;
   1:  PR[GP1:91,2] = PR[GP1:90,2] + -19.115;
   1:L PR[91] R[100]mm/sec CNT100;
   1:  PR[GP1:91,1] = PR[GP1:90,1] + 22.069;
   1:  PR[GP1:91,2] = PR[GP1:90,2] + -19.130;
   1:L PR[91] R[100]mm/sec CNT100;
   1:  PR[GP1:91,1] = PR[GP1:90,1] + 25.028;
   1:  PR[GP1:91,2] = PR[GP1:90,2] + -19.084;
   1:L PR[91] R[100]mm/sec CNT100;
   1:  PR[GP1:91,1] = PR[GP1:90,1] + 28.147;
   1:  PR[GP1:91,2] = PR[GP1:90,2] + -18.526;
   1:L PR[91] R[100]mm/sec CNT100;
   1:  PR[GP1:91,1] = PR[GP1:90,1] + 30.994;
   1:  PR[GP1:91,2] = PR[GP1:90,2] + -17.509;
   1:L PR[91] R[100]mm/sec CNT100;
   1:  PR[GP1:91,1] = PR[GP1:90,1] + 31.082;
   1:  PR[GP1:91,2] = PR[GP1:90,2] + -17.473;
   1:L PR[91] R[100]mm/sec CNT100;
   1:  PR[GP1:91,1] = PR[GP1:90,1] + 33.699;
   1:  PR[GP1:91,2] = PR[GP1:90,2] + -16.019;
   1:L PR[91] R[100]mm/sec CNT100;
   1:  PR[GP1:91,1] = PR[GP1:90,1] + 36.175;
   1:  PR[GP1:91,2] = PR[GP1:90,2] + -14.058;
   1:L PR[91] R[100]mm/sec CNT100;
   1:  PR[GP1:91,1] = PR[GP1:90,1] + 38.201;
   1:  PR[GP1:91,2] = PR[GP1:90,2] + -11.825;
   1:L PR[91] R[100]mm/sec CNT100;
   1:  PR[GP1:91,1] = PR[GP1:90,1] + 38.247;
   1:  PR[GP1:91,2] = PR[GP1:90,2] + -11.764;
   1:L PR[91] R[100]mm/sec CNT100;
   1:  PR[GP1:91,1] = PR[GP1:90,1] + 39.886;
   1:  PR[GP1:91,2] = PR[GP1:90,2] + -9.223;
   1:L PR[91] R[100]mm/sec CNT100;
   1:  PR[GP1:91,1] = PR[GP1:90,1] + 41.138;
   1:  PR[GP1:91,2] = PR[GP1:90,2] + -6.330;
   1:L PR[91] R[100]mm/sec CNT100;
   1:  PR[GP1:91,1] = PR[GP1:90,1] + 41.859;
   1:  PR[GP1:91,2] = PR[GP1:90,2] + -3.451;
   1:L PR[91] R[100]mm/sec CNT100;
   1:  PR[GP1:91,1] = PR[GP1:90,1] + 42.125;
   1:  PR[GP1:91,2] = PR[GP1:90,2] + -0.312;
   1:L PR[91] R[100]mm/sec CNT100;
   1:  PR[GP1:91,1] = PR[GP1:90,1] + 41.859;
   1:  PR[GP1:91,2] = PR[GP1:90,2] + 2.827;
   1:L PR[91] R[100]mm/sec CNT100;
   1:  PR[GP1:91,1] = PR[GP1:90,1] + 41.138;
   1:  PR[GP1:91,2] = PR[GP1:90,2] + 5.706;
   1:L PR[91] R[100]mm/sec CNT100;
   1:  PR[GP1:91,1] = PR[GP1:90,1] + 39.886;
   1:  PR[GP1:91,2] = PR[GP1:90,2] + 8.599;
   1:L PR[91] R[100]mm/sec CNT100;
   1:  PR[GP1:91,1] = PR[GP1:90,1] + 38.247;
   1:  PR[GP1:91,2] = PR[GP1:90,2] + 11.140;
   1:L PR[91] R[100]mm/sec CNT100;
   1:  PR[GP1:91,1] = PR[GP1:90,1] + 38.201;
   1:  PR[GP1:91,2] = PR[GP1:90,2] + 11.201;
   1:L PR[91] R[100]mm/sec CNT100;
   1:  PR[GP1:91,1] = PR[GP1:90,1] + 36.175;
   1:  PR[GP1:91,2] = PR[GP1:90,2] + 13.435;
   1:L PR[91] R[100]mm/sec CNT100;
   1:  PR[GP1:91,1] = PR[GP1:90,1] + 33.699;
   1:  PR[GP1:91,2] = PR[GP1:90,2] + 15.395;
   1:L PR[91] R[100]mm/sec CNT100;
   1:  PR[GP1:91,1] = PR[GP1:90,1] + 31.082;
   1:  PR[GP1:91,2] = PR[GP1:90,2] + 16.848;
   1:L PR[91] R[100]mm/sec CNT100;
   1:  PR[GP1:91,1] = PR[GP1:90,1] + 30.994;
   1:  PR[GP1:91,2] = PR[GP1:90,2] + 16.885;
   1:L PR[91] R[100]mm/sec CNT100;
   1:  PR[GP1:91,1] = PR[GP1:90,1] + 28.147;
   1:  PR[GP1:91,2] = PR[GP1:90,2] + 17.902;
   1:L PR[91] R[100]mm/sec CNT100;
   1:  PR[GP1:91,1] = PR[GP1:90,1] + 25.028;
   1:  PR[GP1:91,2] = PR[GP1:90,2] + 18.460;
   1:L PR[91] R[100]mm/sec CNT100;
   1:  PR[GP1:91,1] = PR[GP1:90,1] + 22.087;
   1:  PR[GP1:91,2] = PR[GP1:90,2] + 18.506;
   1:L PR[91] R[100]mm/sec CNT100;
   1:  PR[GP1:91,1] = PR[GP1:90,1] + 18.950;
   1:  PR[GP1:91,2] = PR[GP1:90,2] + 18.045;
   1:L PR[91] R[100]mm/sec CNT100;
   1:  PR[GP1:91,1] = PR[GP1:90,1] + 16.100;
   1:  PR[GP1:91,2] = PR[GP1:90,2] + 17.127;
   1:L PR[91] R[100]mm/sec CNT100;
   1:  PR[GP1:91,1] = PR[GP1:90,1] + 15.972;
   1:  PR[GP1:91,2] = PR[GP1:90,2] + 17.075;
   1:L PR[91] R[100]mm/sec CNT100;
   1:  PR[GP1:91,1] = PR[GP1:90,1] + 13.334;
   1:  PR[GP1:91,2] = PR[GP1:90,2] + 15.718;
   1:L PR[91] R[100]mm/sec CNT100;
   1:  PR[GP1:91,1] = PR[GP1:90,1] + 10.778;
   1:  PR[GP1:91,2] = PR[GP1:90,2] + 13.818;
   1:L PR[91] R[100]mm/sec CNT100;
   1:  PR[GP1:91,1] = PR[GP1:90,1] + 8.726;
   1:  PR[GP1:91,2] = PR[GP1:90,2] + 11.694;
   1:L PR[91] R[100]mm/sec CNT100;
   1:  PR[GP1:91,1] = PR[GP1:90,1] + 8.619;
   1:  PR[GP1:91,2] = PR[GP1:90,2] + 11.558;
   1:L PR[91] R[100]mm/sec CNT100;
   1:  PR[GP1:91,1] = PR[GP1:90,1] + 6.932;
   1:  PR[GP1:91,2] = PR[GP1:90,2] + 9.116;
   1:L PR[91] R[100]mm/sec CNT100;
   1:  PR[GP1:91,1] = PR[GP1:90,1] + 5.654;
   1:  PR[GP1:91,2] = PR[GP1:90,2] + 6.407;
   1:L PR[91] R[100]mm/sec CNT100;
   1:  PR[GP1:91,1] = PR[GP1:90,1] + 5.583;
   1:  PR[GP1:91,2] = PR[GP1:90,2] + 6.245;
   1:L PR[91] R[100]mm/sec CNT100;
   1:  PR[GP1:91,1] = PR[GP1:90,1] + 4.901;
   1:  PR[GP1:91,2] = PR[GP1:90,2] + 3.847;
   1:L PR[91] R[100]mm/sec CNT100;
   1:  PR[GP1:91,1] = PR[GP1:90,1] + 4.940;
   1:  PR[GP1:91,2] = PR[GP1:90,2] + 3.764;
   1:L PR[91] R[100]mm/sec CNT100;
   1:  PR[GP1:91,1] = PR[GP1:90,1] + 4.415;
   1:  PR[GP1:91,2] = PR[GP1:90,2] + 2.372;
   1:L PR[91] R[100]mm/sec CNT100;
   1:  PR[GP1:91,1] = PR[GP1:90,1] + 3.692;
   1:  PR[GP1:91,2] = PR[GP1:90,2] + 1.522;
   1:L PR[91] R[100]mm/sec CNT100;
   1:  PR[GP1:91,1] = PR[GP1:90,1] + 2.804;
   1:  PR[GP1:91,2] = PR[GP1:90,2] + 1.025;
   1:L PR[91] R[100]mm/sec CNT100;
   1:  PR[GP1:91,1] = PR[GP1:90,1] + 2.393;
   1:  PR[GP1:91,2] = PR[GP1:90,2] + 0.903;
   1:L PR[91] R[100]mm/sec CNT100;
   1:  PR[GP1:91,1] = PR[GP1:90,1] + 1.770;
   1:  PR[GP1:91,2] = PR[GP1:90,2] + 0.795;
   1:L PR[91] R[100]mm/sec CNT100;
   1:  PR[GP1:91,1] = PR[GP1:90,1] + -1.614;
   1:  PR[GP1:91,2] = PR[GP1:90,2] + 0.798;
   1:L PR[91] R[100]mm/sec CNT100;
   1:  PR[91] = PR[90];
   1:  PR[GP1:91,1] = PR[GP1:90,1] + -2.635;
   1:  PR[GP1:91,2] = PR[GP1:90,2] + 1.180;
   1:  PR[GP1:91,3] = PR[GP1:90,3] + 5.795;
   1:L PR[91] R[100]mm/sec CNT100;
   1:  PR[GP1:91,1] = PR[GP1:90,1] + -3.599;
   1:  PR[GP1:91,2] = PR[GP1:90,2] + 1.759;
   1:L PR[91] R[100]mm/sec CNT100;
   1:  PR[GP1:91,1] = PR[GP1:90,1] + -4.311;
   1:  PR[GP1:91,2] = PR[GP1:90,2] + 2.660;
   1:L PR[91] R[100]mm/sec CNT100;
   1:  PR[GP1:91,1] = PR[GP1:90,1] + -4.617;
   1:  PR[GP1:91,2] = PR[GP1:90,2] + 3.508;
   1:L PR[91] R[100]mm/sec CNT100;
   1:  PR[GP1:91,1] = PR[GP1:90,1] + -5.291;
   1:  PR[GP1:91,2] = PR[GP1:90,2] + 5.952;
   1:L PR[91] R[100]mm/sec CNT100;
   1:  PR[GP1:91,1] = PR[GP1:90,1] + -6.352;
   1:  PR[GP1:91,2] = PR[GP1:90,2] + 8.203;
   1:L PR[91] R[100]mm/sec CNT100;
   1:  PR[GP1:91,1] = PR[GP1:90,1] + -6.773;
   1:  PR[GP1:91,2] = PR[GP1:90,2] + 9.186;
   1:L PR[91] R[100]mm/sec CNT100;
   1:  PR[GP1:91,1] = PR[GP1:90,1] + -8.175;
   1:  PR[GP1:91,2] = PR[GP1:90,2] + 11.216;
   1:L PR[91] R[100]mm/sec CNT100;
   1:  PR[GP1:91,1] = PR[GP1:90,1] + -8.741;
   1:  PR[GP1:91,2] = PR[GP1:90,2] + 11.930;
   1:L PR[91] R[100]mm/sec CNT100;
   1:  PR[GP1:91,1] = PR[GP1:90,1] + -10.481;
   1:  PR[GP1:91,2] = PR[GP1:90,2] + 13.731;
   1:L PR[91] R[100]mm/sec CNT100;
   1:  PR[GP1:91,1] = PR[GP1:90,1] + -13.246;
   1:  PR[GP1:91,2] = PR[GP1:90,2] + 15.785;
   1:L PR[91] R[100]mm/sec CNT100;
   1:  PR[GP1:91,1] = PR[GP1:90,1] + -15.507;
   1:  PR[GP1:91,2] = PR[GP1:90,2] + 16.949;
   1:L PR[91] R[100]mm/sec CNT100;
   1:  PR[GP1:91,1] = PR[GP1:90,1] + -16.240;
   1:  PR[GP1:91,2] = PR[GP1:90,2] + 17.242;
   1:L PR[91] R[100]mm/sec CNT100;
   1:  PR[GP1:91,1] = PR[GP1:90,1] + -18.715;
   1:  PR[GP1:91,2] = PR[GP1:90,2] + 18.039;
   1:L PR[91] R[100]mm/sec CNT100;
   1:  PR[GP1:91,1] = PR[GP1:90,1] + -21.316;
   1:  PR[GP1:91,2] = PR[GP1:90,2] + 18.427;
   1:L PR[91] R[100]mm/sec CNT100;
   1:  PR[GP1:91,1] = PR[GP1:90,1] + -22.055;
   1:  PR[GP1:91,2] = PR[GP1:90,2] + 18.516;
   1:L PR[91] R[100]mm/sec CNT100;
   1:  PR[GP1:91,1] = PR[GP1:90,1] + -24.642;
   1:  PR[GP1:91,2] = PR[GP1:90,2] + 18.476;
   1:L PR[91] R[100]mm/sec CNT100;
   1:  PR[GP1:91,1] = PR[GP1:90,1] + -27.312;
   1:  PR[GP1:91,2] = PR[GP1:90,2] + 17.991;
   1:L PR[91] R[100]mm/sec CNT100;
   1:  PR[GP1:91,1] = PR[GP1:90,1] + -28.007;
   1:  PR[GP1:91,2] = PR[GP1:90,2] + 17.893;
   1:L PR[91] R[100]mm/sec CNT100;
   1:  PR[GP1:91,1] = PR[GP1:90,1] + -30.502;
   1:  PR[GP1:91,2] = PR[GP1:90,2] + 17.002;
   1:L PR[91] R[100]mm/sec CNT100;
   1:  PR[GP1:91,1] = PR[GP1:90,1] + -31.088;
   1:  PR[GP1:91,2] = PR[GP1:90,2] + 16.755;
   1:L PR[91] R[100]mm/sec CNT100;
   1:  PR[GP1:91,1] = PR[GP1:90,1] + -33.420;
   1:  PR[GP1:91,2] = PR[GP1:90,2] + 15.460;
   1:L PR[91] R[100]mm/sec CNT100;
   1:  PR[GP1:91,1] = PR[GP1:90,1] + -36.049;
   1:  PR[GP1:91,2] = PR[GP1:90,2] + 13.385;
   1:L PR[91] R[100]mm/sec CNT100;
   1:  PR[GP1:91,1] = PR[GP1:90,1] + -37.863;
   1:  PR[GP1:91,2] = PR[GP1:90,2] + 11.385;
   1:L PR[91] R[100]mm/sec CNT100;
   1:  PR[GP1:91,1] = PR[GP1:90,1] + -38.207;
   1:  PR[GP1:91,2] = PR[GP1:90,2] + 10.934;
   1:L PR[91] R[100]mm/sec CNT100;
   1:  PR[GP1:91,1] = PR[GP1:90,1] + -39.681;
   1:  PR[GP1:91,2] = PR[GP1:90,2] + 8.650;
   1:L PR[91] R[100]mm/sec CNT100;
   1:  PR[GP1:91,1] = PR[GP1:90,1] + -40.995;
   1:  PR[GP1:91,2] = PR[GP1:90,2] + 5.592;
   1:L PR[91] R[100]mm/sec CNT100;
   1:  PR[GP1:91,1] = PR[GP1:90,1] + -41.644;
   1:  PR[GP1:91,2] = PR[GP1:90,2] + 3.002;
   1:L PR[91] R[100]mm/sec CNT100;
   1:  PR[GP1:91,1] = PR[GP1:90,1] + -41.874;
   1:  PR[GP1:91,2] = PR[GP1:90,2] + 0.192;
   1:L PR[91] R[100]mm/sec CNT100;
   1:  PR[GP1:91,1] = PR[GP1:90,1] + -41.944;
   1:  PR[GP1:91,2] = PR[GP1:90,2] + -0.346;
   1:L PR[91] R[100]mm/sec CNT100;
   1:  PR[GP1:91,1] = PR[GP1:90,1] + -41.721;
   1:  PR[GP1:91,2] = PR[GP1:90,2] + -3.067;
   1:L PR[91] R[100]mm/sec CNT100;
   1:  PR[GP1:91,1] = PR[GP1:90,1] + -41.652;
   1:  PR[GP1:91,2] = PR[GP1:90,2] + -3.592;
   1:L PR[91] R[100]mm/sec CNT100;
   1:  PR[GP1:91,1] = PR[GP1:90,1] + -40.995;
   1:  PR[GP1:91,2] = PR[GP1:90,2] + -6.216;
   1:L PR[91] R[100]mm/sec CNT100;
   1:  PR[GP1:91,1] = PR[GP1:90,1] + -39.681;
   1:  PR[GP1:91,2] = PR[GP1:90,2] + -9.274;
   1:L PR[91] R[100]mm/sec CNT100;
   1:  PR[GP1:91,1] = PR[GP1:90,1] + -38.207;
   1:  PR[GP1:91,2] = PR[GP1:90,2] + -11.558;
   1:L PR[91] R[100]mm/sec CNT100;
   1:  PR[GP1:91,1] = PR[GP1:90,1] + -37.863;
   1:  PR[GP1:91,2] = PR[GP1:90,2] + -12.009;
   1:L PR[91] R[100]mm/sec CNT100;
   1:  PR[GP1:91,1] = PR[GP1:90,1] + -36.049;
   1:  PR[GP1:91,2] = PR[GP1:90,2] + -14.009;
   1:L PR[91] R[100]mm/sec CNT100;
   1:  PR[GP1:91,1] = PR[GP1:90,1] + -33.420;
   1:  PR[GP1:91,2] = PR[GP1:90,2] + -16.084;
   1:L PR[91] R[100]mm/sec CNT100;
   1:  PR[GP1:91,1] = PR[GP1:90,1] + -31.088;
   1:  PR[GP1:91,2] = PR[GP1:90,2] + -17.379;
   1:L PR[91] R[100]mm/sec CNT100;
   1:  PR[GP1:91,1] = PR[GP1:90,1] + -30.501;
   1:  PR[GP1:91,2] = PR[GP1:90,2] + -17.626;
   1:L PR[91] R[100]mm/sec CNT100;
   1:  PR[GP1:91,1] = PR[GP1:90,1] + -27.981;
   1:  PR[GP1:91,2] = PR[GP1:90,2] + -18.526;
   1:L PR[91] R[100]mm/sec CNT100;
   1:  PR[GP1:91,1] = PR[GP1:90,1] + -25.336;
   1:  PR[GP1:91,2] = PR[GP1:90,2] + -19.006;
   1:L PR[91] R[100]mm/sec CNT100;
   1:  PR[GP1:91,1] = PR[GP1:90,1] + -24.672;
   1:  PR[GP1:91,2] = PR[GP1:90,2] + -19.099;
   1:L PR[91] R[100]mm/sec CNT100;
   1:  PR[GP1:91,1] = PR[GP1:90,1] + -22.075;
   1:  PR[GP1:91,2] = PR[GP1:90,2] + -19.140;
   1:L PR[91] R[100]mm/sec CNT100;
   1:  PR[GP1:91,1] = PR[GP1:90,1] + -19.398;
   1:  PR[GP1:91,2] = PR[GP1:90,2] + -18.741;
   1:L PR[91] R[100]mm/sec CNT100;
   1:  PR[GP1:91,1] = PR[GP1:90,1] + -18.695;
   1:  PR[GP1:91,2] = PR[GP1:90,2] + -18.657;
   1:L PR[91] R[100]mm/sec CNT100;
   1:  PR[GP1:91,1] = PR[GP1:90,1] + -16.240;
   1:  PR[GP1:91,2] = PR[GP1:90,2] + -17.866;
   1:L PR[91] R[100]mm/sec CNT100;
   1:  PR[GP1:91,1] = PR[GP1:90,1] + -15.507;
   1:  PR[GP1:91,2] = PR[GP1:90,2] + -17.573;
   1:L PR[91] R[100]mm/sec CNT100;
   1:  PR[GP1:91,1] = PR[GP1:90,1] + -13.246;
   1:  PR[GP1:91,2] = PR[GP1:90,2] + -16.409;
   1:L PR[91] R[100]mm/sec CNT100;
   1:  PR[GP1:91,1] = PR[GP1:90,1] + -10.481;
   1:  PR[GP1:91,2] = PR[GP1:90,2] + -14.355;
   1:L PR[91] R[100]mm/sec CNT100;
   1:  PR[GP1:91,1] = PR[GP1:90,1] + -8.742;
   1:  PR[GP1:91,2] = PR[GP1:90,2] + -12.554;
   1:L PR[91] R[100]mm/sec CNT100;
   1:  PR[GP1:91,1] = PR[GP1:90,1] + -8.175;
   1:  PR[GP1:91,2] = PR[GP1:90,2] + -11.840;
   1:L PR[91] R[100]mm/sec CNT100;
   1:  PR[GP1:91,1] = PR[GP1:90,1] + -6.758;
   1:  PR[GP1:91,2] = PR[GP1:90,2] + -9.788;
   1:L PR[91] R[100]mm/sec CNT100;
   1:  PR[GP1:91,1] = PR[GP1:90,1] + -5.683;
   1:  PR[GP1:91,2] = PR[GP1:90,2] + -7.510;
   1:L PR[91] R[100]mm/sec CNT100;
   1:  PR[GP1:91,1] = PR[GP1:90,1] + -5.305;
   1:  PR[GP1:91,2] = PR[GP1:90,2] + -6.641;
   1:L PR[91] R[100]mm/sec CNT100;
   1:  PR[GP1:91,1] = PR[GP1:90,1] + -4.800;
   1:  PR[GP1:91,2] = PR[GP1:90,2] + -4.862;
   1:L PR[91] R[100]mm/sec CNT100;
   1:  PR[GP1:91,1] = PR[GP1:90,1] + -4.851;
   1:  PR[GP1:91,2] = PR[GP1:90,2] + -4.789;
   1:L PR[91] R[100]mm/sec CNT100;
   1:  PR[GP1:91,1] = PR[GP1:90,1] + -4.310;
   1:  PR[GP1:91,2] = PR[GP1:90,2] + -3.282;
   1:L PR[91] R[100]mm/sec CNT100;
   1:  PR[GP1:91,1] = PR[GP1:90,1] + -3.599;
   1:  PR[GP1:91,2] = PR[GP1:90,2] + -2.383;
   1:L PR[91] R[100]mm/sec CNT100;
   1:  PR[GP1:91,1] = PR[GP1:90,1] + -2.635;
   1:  PR[GP1:91,2] = PR[GP1:90,2] + -1.804;
   1:L PR[91] R[100]mm/sec CNT100;
   1:  PR[GP1:91,1] = PR[GP1:90,1] + -1.658;
   1:  PR[GP1:91,2] = PR[GP1:90,2] + -1.607;
   1:L PR[91] R[100]mm/sec CNT100;
   1:  PR[GP1:91,1] = PR[GP1:90,1] + 1.815;
   1:L PR[91] R[100]mm/sec CNT100;
   1:  PR[GP1:91,1] = PR[GP1:90,1] + 2.792;
   1:  PR[GP1:91,2] = PR[GP1:90,2] + -1.804;
   1:L PR[91] R[100]mm/sec CNT100;
   1:  PR[GP1:91,1] = PR[GP1:90,1] + 3.756;
   1:  PR[GP1:91,2] = PR[GP1:90,2] + -2.383;
   1:L PR[91] R[100]mm/sec CNT100;
   1:  PR[GP1:91,1] = PR[GP1:90,1] + 4.467;
   1:  PR[GP1:91,2] = PR[GP1:90,2] + -3.284;
   1:L PR[91] R[100]mm/sec CNT100;
   1:  PR[GP1:91,1] = PR[GP1:90,1] + 4.773;
   1:  PR[GP1:91,2] = PR[GP1:90,2] + -4.132;
   1:L PR[91] R[100]mm/sec CNT100;
   1:  PR[GP1:91,1] = PR[GP1:90,1] + 5.450;
   1:  PR[GP1:91,2] = PR[GP1:90,2] + -6.586;
   1:L PR[91] R[100]mm/sec CNT100;
   1:  PR[GP1:91,1] = PR[GP1:90,1] + 6.515;
   1:  PR[GP1:91,2] = PR[GP1:90,2] + -8.844;
   1:L PR[91] R[100]mm/sec CNT100;
   1:  PR[GP1:91,1] = PR[GP1:90,1] + 6.929;
   1:  PR[GP1:91,2] = PR[GP1:90,2] + -9.808;
   1:L PR[91] R[100]mm/sec CNT100;
   1:  PR[GP1:91,1] = PR[GP1:90,1] + 8.332;
   1:  PR[GP1:91,2] = PR[GP1:90,2] + -11.840;
   1:L PR[91] R[100]mm/sec CNT100;
   1:  PR[GP1:91,1] = PR[GP1:90,1] + 8.898;
   1:  PR[GP1:91,2] = PR[GP1:90,2] + -12.554;
   1:L PR[91] R[100]mm/sec CNT100;
   1:  PR[GP1:91,1] = PR[GP1:90,1] + 10.637;
   1:  PR[GP1:91,2] = PR[GP1:90,2] + -14.355;
   1:L PR[91] R[100]mm/sec CNT100;
   1:  PR[GP1:91,1] = PR[GP1:90,1] + 13.402;
   1:  PR[GP1:91,2] = PR[GP1:90,2] + -16.409;
   1:L PR[91] R[100]mm/sec CNT100;
   1:  PR[GP1:91,1] = PR[GP1:90,1] + 15.664;
   1:  PR[GP1:91,2] = PR[GP1:90,2] + -17.573;
   1:L PR[91] R[100]mm/sec CNT100;
   1:  PR[GP1:91,1] = PR[GP1:90,1] + 16.396;
   1:  PR[GP1:91,2] = PR[GP1:90,2] + -17.866;
   1:L PR[91] R[100]mm/sec CNT100;
   1:  PR[GP1:91,1] = PR[GP1:90,1] + 18.871;
   1:  PR[GP1:91,2] = PR[GP1:90,2] + -18.663;
   1:L PR[91] R[100]mm/sec CNT100;
   1:  PR[GP1:91,1] = PR[GP1:90,1] + 21.472;
   1:  PR[GP1:91,2] = PR[GP1:90,2] + -19.051;
   1:L PR[91] R[100]mm/sec CNT100;
   1:  PR[GP1:91,1] = PR[GP1:90,1] + 22.212;
   1:  PR[GP1:91,2] = PR[GP1:90,2] + -19.140;
   1:L PR[91] R[100]mm/sec CNT100;
   1:  PR[GP1:91,1] = PR[GP1:90,1] + 24.799;
   1:  PR[GP1:91,2] = PR[GP1:90,2] + -19.100;
   1:L PR[91] R[100]mm/sec CNT100;
   1:  PR[GP1:91,1] = PR[GP1:90,1] + 27.469;
   1:  PR[GP1:91,2] = PR[GP1:90,2] + -18.615;
   1:L PR[91] R[100]mm/sec CNT100;
   1:  PR[GP1:91,1] = PR[GP1:90,1] + 28.164;
   1:  PR[GP1:91,2] = PR[GP1:90,2] + -18.517;
   1:L PR[91] R[100]mm/sec CNT100;
   1:  PR[GP1:91,1] = PR[GP1:90,1] + 30.658;
   1:  PR[GP1:91,2] = PR[GP1:90,2] + -17.626;
   1:L PR[91] R[100]mm/sec CNT100;
   1:  PR[GP1:91,1] = PR[GP1:90,1] + 31.245;
   1:  PR[GP1:91,2] = PR[GP1:90,2] + -17.379;
   1:L PR[91] R[100]mm/sec CNT100;
   1:  PR[GP1:91,1] = PR[GP1:90,1] + 33.576;
   1:  PR[GP1:91,2] = PR[GP1:90,2] + -16.084;
   1:L PR[91] R[100]mm/sec CNT100;
   1:  PR[GP1:91,1] = PR[GP1:90,1] + 36.206;
   1:  PR[GP1:91,2] = PR[GP1:90,2] + -14.009;
   1:L PR[91] R[100]mm/sec CNT100;
   1:  PR[GP1:91,1] = PR[GP1:90,1] + 38.019;
   1:  PR[GP1:91,2] = PR[GP1:90,2] + -12.009;
   1:L PR[91] R[100]mm/sec CNT100;
   1:  PR[GP1:91,1] = PR[GP1:90,1] + 38.364;
   1:  PR[GP1:91,2] = PR[GP1:90,2] + -11.558;
   1:L PR[91] R[100]mm/sec CNT100;
   1:  PR[GP1:91,1] = PR[GP1:90,1] + 39.837;
   1:  PR[GP1:91,2] = PR[GP1:90,2] + -9.273;
   1:L PR[91] R[100]mm/sec CNT100;
   1:  PR[GP1:91,1] = PR[GP1:90,1] + 41.152;
   1:  PR[GP1:91,2] = PR[GP1:90,2] + -6.216;
   1:L PR[91] R[100]mm/sec CNT100;
   1:  PR[GP1:91,1] = PR[GP1:90,1] + 41.801;
   1:  PR[GP1:91,2] = PR[GP1:90,2] + -3.626;
   1:L PR[91] R[100]mm/sec CNT100;
   1:  PR[GP1:91,1] = PR[GP1:90,1] + 42.031;
   1:  PR[GP1:91,2] = PR[GP1:90,2] + -0.816;
   1:L PR[91] R[100]mm/sec CNT100;
   1:  PR[GP1:91,1] = PR[GP1:90,1] + 42.101;
   1:  PR[GP1:91,2] = PR[GP1:90,2] + -0.278;
   1:L PR[91] R[100]mm/sec CNT100;
   1:  PR[GP1:91,1] = PR[GP1:90,1] + 41.878;
   1:  PR[GP1:91,2] = PR[GP1:90,2] + 2.443;
   1:L PR[91] R[100]mm/sec CNT100;
   1:  PR[GP1:91,1] = PR[GP1:90,1] + 41.809;
   1:  PR[GP1:91,2] = PR[GP1:90,2] + 2.969;
   1:L PR[91] R[100]mm/sec CNT100;
   1:  PR[GP1:91,1] = PR[GP1:90,1] + 41.152;
   1:  PR[GP1:91,2] = PR[GP1:90,2] + 5.592;
   1:L PR[91] R[100]mm/sec CNT100;
   1:  PR[GP1:91,1] = PR[GP1:90,1] + 39.837;
   1:  PR[GP1:91,2] = PR[GP1:90,2] + 8.650;
   1:L PR[91] R[100]mm/sec CNT100;
   1:  PR[GP1:91,1] = PR[GP1:90,1] + 38.364;
   1:  PR[GP1:91,2] = PR[GP1:90,2] + 10.934;
   1:L PR[91] R[100]mm/sec CNT100;
   1:  PR[GP1:91,1] = PR[GP1:90,1] + 38.019;
   1:  PR[GP1:91,2] = PR[GP1:90,2] + 11.386;
   1:L PR[91] R[100]mm/sec CNT100;
   1:  PR[GP1:91,1] = PR[GP1:90,1] + 36.205;
   1:  PR[GP1:91,2] = PR[GP1:90,2] + 13.386;
   1:L PR[91] R[100]mm/sec CNT100;
   1:  PR[GP1:91,1] = PR[GP1:90,1] + 33.576;
   1:  PR[GP1:91,2] = PR[GP1:90,2] + 15.461;
   1:L PR[91] R[100]mm/sec CNT100;
   1:  PR[GP1:91,1] = PR[GP1:90,1] + 31.245;
   1:  PR[GP1:91,2] = PR[GP1:90,2] + 16.755;
   1:L PR[91] R[100]mm/sec CNT100;
   1:  PR[GP1:91,1] = PR[GP1:90,1] + 30.658;
   1:  PR[GP1:91,2] = PR[GP1:90,2] + 17.002;
   1:L PR[91] R[100]mm/sec CNT100;
   1:  PR[GP1:91,1] = PR[GP1:90,1] + 28.136;
   1:  PR[GP1:91,2] = PR[GP1:90,2] + 17.903;
   1:L PR[91] R[100]mm/sec CNT100;
   1:  PR[GP1:91,1] = PR[GP1:90,1] + 25.492;
   1:  PR[GP1:91,2] = PR[GP1:90,2] + 18.382;
   1:L PR[91] R[100]mm/sec CNT100;
   1:  PR[GP1:91,1] = PR[GP1:90,1] + 24.827;
   1:  PR[GP1:91,2] = PR[GP1:90,2] + 18.475;
   1:L PR[91] R[100]mm/sec CNT100;
   1:  PR[GP1:91,1] = PR[GP1:90,1] + 22.231;
   1:  PR[GP1:91,2] = PR[GP1:90,2] + 18.516;
   1:L PR[91] R[100]mm/sec CNT100;
   1:  PR[GP1:91,1] = PR[GP1:90,1] + 19.554;
   1:  PR[GP1:91,2] = PR[GP1:90,2] + 18.117;
   1:L PR[91] R[100]mm/sec CNT100;
   1:  PR[GP1:91,1] = PR[GP1:90,1] + 18.850;
   1:  PR[GP1:91,2] = PR[GP1:90,2] + 18.032;
   1:L PR[91] R[100]mm/sec CNT100;
   1:  PR[GP1:91,1] = PR[GP1:90,1] + 16.395;
   1:  PR[GP1:91,2] = PR[GP1:90,2] + 17.242;
   1:L PR[91] R[100]mm/sec CNT100;
   1:  PR[GP1:91,1] = PR[GP1:90,1] + 15.662;
   1:  PR[GP1:91,2] = PR[GP1:90,2] + 16.948;
   1:L PR[91] R[100]mm/sec CNT100;
   1:  PR[GP1:91,1] = PR[GP1:90,1] + 13.401;
   1:  PR[GP1:91,2] = PR[GP1:90,2] + 15.784;
   1:L PR[91] R[100]mm/sec CNT100;
   1:  PR[GP1:91,1] = PR[GP1:90,1] + 10.636;
   1:  PR[GP1:91,2] = PR[GP1:90,2] + 13.729;
   1:L PR[91] R[100]mm/sec CNT100;
   1:  PR[GP1:91,1] = PR[GP1:90,1] + 8.897;
   1:  PR[GP1:91,2] = PR[GP1:90,2] + 11.929;
   1:L PR[91] R[100]mm/sec CNT100;
   1:  PR[GP1:91,1] = PR[GP1:90,1] + 8.331;
   1:  PR[GP1:91,2] = PR[GP1:90,2] + 11.214;
   1:L PR[91] R[100]mm/sec CNT100;
   1:  PR[GP1:91,1] = PR[GP1:90,1] + 6.914;
   1:  PR[GP1:91,2] = PR[GP1:90,2] + 9.162;
   1:L PR[91] R[100]mm/sec CNT100;
   1:  PR[GP1:91,1] = PR[GP1:90,1] + 5.838;
   1:  PR[GP1:91,2] = PR[GP1:90,2] + 6.881;
   1:L PR[91] R[100]mm/sec CNT100;
   1:  PR[GP1:91,1] = PR[GP1:90,1] + 5.465;
   1:  PR[GP1:91,2] = PR[GP1:90,2] + 6.033;
   1:L PR[91] R[100]mm/sec CNT100;
   1:  PR[GP1:91,1] = PR[GP1:90,1] + 4.959;
   1:  PR[GP1:91,2] = PR[GP1:90,2] + 4.253;
   1:L PR[91] R[100]mm/sec CNT100;
   1:  PR[GP1:91,1] = PR[GP1:90,1] + 5.012;
   1:  PR[GP1:91,2] = PR[GP1:90,2] + 4.181;
   1:L PR[91] R[100]mm/sec CNT100;
   1:  PR[GP1:91,1] = PR[GP1:90,1] + 4.466;
   1:  PR[GP1:91,2] = PR[GP1:90,2] + 2.658;
   1:L PR[91] R[100]mm/sec CNT100;
   1:  PR[GP1:91,1] = PR[GP1:90,1] + 3.755;
   1:  PR[GP1:91,2] = PR[GP1:90,2] + 1.758;
   1:L PR[91] R[100]mm/sec CNT100;
   1:  PR[GP1:91,1] = PR[GP1:90,1] + 2.792;
   1:  PR[GP1:91,2] = PR[GP1:90,2] + 1.180;
   1:L PR[91] R[100]mm/sec CNT100;
   1:  PR[GP1:91,1] = PR[GP1:90,1] + 1.815;
   1:  PR[GP1:91,2] = PR[GP1:90,2] + 0.983;
   1:L PR[91] R[100]mm/sec CNT100;
   1:  PR[GP1:91,1] = PR[GP1:90,1] + -1.658;
   1:L PR[91] R[100]mm/sec CNT100;
   1:  PR[91] = PR[90];
   1:  PR[GP1:91,1] = PR[GP1:90,1] + -2.659;
   1:  PR[GP1:91,2] = PR[GP1:90,2] + 1.452;
   1:  PR[GP1:91,3] = PR[GP1:90,3] + 6.405;
   1:L PR[91] R[100]mm/sec CNT100;
   1:  PR[GP1:91,1] = PR[GP1:90,1] + -3.620;
   1:  PR[GP1:91,2] = PR[GP1:90,2] + 2.064;
   1:L PR[91] R[100]mm/sec CNT100;
   1:  PR[GP1:91,1] = PR[GP1:90,1] + -4.368;
   1:  PR[GP1:91,2] = PR[GP1:90,2] + 3.035;
   1:L PR[91] R[100]mm/sec CNT100;
   1:  PR[GP1:91,1] = PR[GP1:90,1] + -4.629;
   1:  PR[GP1:91,2] = PR[GP1:90,2] + 3.758;
   1:L PR[91] R[100]mm/sec CNT100;
   1:  PR[GP1:91,1] = PR[GP1:90,1] + -5.162;
   1:  PR[GP1:91,2] = PR[GP1:90,2] + 5.691;
   1:L PR[91] R[100]mm/sec CNT100;
   1:  PR[GP1:91,1] = PR[GP1:90,1] + -5.999;
   1:  PR[GP1:91,2] = PR[GP1:90,2] + 7.466;
   1:L PR[91] R[100]mm/sec CNT100;
   1:  PR[GP1:91,1] = PR[GP1:90,1] + -6.755;
   1:  PR[GP1:91,2] = PR[GP1:90,2] + 9.233;
   1:L PR[91] R[100]mm/sec CNT100;
   1:  PR[GP1:91,1] = PR[GP1:90,1] + -7.888;
   1:  PR[GP1:91,2] = PR[GP1:90,2] + 10.873;
   1:L PR[91] R[100]mm/sec CNT100;
   1:  PR[GP1:91,1] = PR[GP1:90,1] + -8.914;
   1:  PR[GP1:91,2] = PR[GP1:90,2] + 12.166;
   1:L PR[91] R[100]mm/sec CNT100;
   1:  PR[GP1:91,1] = PR[GP1:90,1] + -10.340;
   1:  PR[GP1:91,2] = PR[GP1:90,2] + 13.643;
   1:L PR[91] R[100]mm/sec CNT100;
   1:  PR[GP1:91,1] = PR[GP1:90,1] + -13.314;
   1:  PR[GP1:91,2] = PR[GP1:90,2] + 15.853;
   1:L PR[91] R[100]mm/sec CNT100;
   1:  PR[GP1:91,1] = PR[GP1:90,1] + -15.199;
   1:  PR[GP1:91,2] = PR[GP1:90,2] + 16.823;
   1:L PR[91] R[100]mm/sec CNT100;
   1:  PR[GP1:91,1] = PR[GP1:90,1] + -16.535;
   1:  PR[GP1:91,2] = PR[GP1:90,2] + 17.357;
   1:L PR[91] R[100]mm/sec CNT100;
   1:  PR[GP1:91,1] = PR[GP1:90,1] + -18.634;
   1:  PR[GP1:91,2] = PR[GP1:90,2] + 18.033;
   1:L PR[91] R[100]mm/sec CNT100;
   1:  PR[GP1:91,1] = PR[GP1:90,1] + -20.844;
   1:  PR[GP1:91,2] = PR[GP1:90,2] + 18.363;
   1:L PR[91] R[100]mm/sec CNT100;
   1:  PR[GP1:91,1] = PR[GP1:90,1] + -22.198;
   1:  PR[GP1:91,2] = PR[GP1:90,2] + 18.526;
   1:L PR[91] R[100]mm/sec CNT100;
   1:  PR[GP1:91,1] = PR[GP1:90,1] + -24.415;
   1:  PR[GP1:91,2] = PR[GP1:90,2] + 18.491;
   1:L PR[91] R[100]mm/sec CNT100;
   1:  PR[GP1:91,1] = PR[GP1:90,1] + -26.721;
   1:  PR[GP1:91,2] = PR[GP1:90,2] + 18.073;
   1:L PR[91] R[100]mm/sec CNT100;
   1:  PR[GP1:91,1] = PR[GP1:90,1] + -27.999;
   1:  PR[GP1:91,2] = PR[GP1:90,2] + 17.892;
   1:L PR[91] R[100]mm/sec CNT100;
   1:  PR[GP1:91,1] = PR[GP1:90,1] + -30.166;
   1:  PR[GP1:91,2] = PR[GP1:90,2] + 17.118;
   1:L PR[91] R[100]mm/sec CNT100;
   1:  PR[GP1:91,1] = PR[GP1:90,1] + -31.252;
   1:  PR[GP1:91,2] = PR[GP1:90,2] + 16.661;
   1:L PR[91] R[100]mm/sec CNT100;
   1:  PR[GP1:91,1] = PR[GP1:90,1] + -33.297;
   1:  PR[GP1:91,2] = PR[GP1:90,2] + 15.526;
   1:L PR[91] R[100]mm/sec CNT100;
   1:  PR[GP1:91,1] = PR[GP1:90,1] + -36.079;
   1:  PR[GP1:91,2] = PR[GP1:90,2] + 13.336;
   1:L PR[91] R[100]mm/sec CNT100;
   1:  PR[GP1:91,1] = PR[GP1:90,1] + -37.681;
   1:  PR[GP1:91,2] = PR[GP1:90,2] + 11.570;
   1:L PR[91] R[100]mm/sec CNT100;
   1:  PR[GP1:91,1] = PR[GP1:90,1] + -38.324;
   1:  PR[GP1:91,2] = PR[GP1:90,2] + 10.727;
   1:L PR[91] R[100]mm/sec CNT100;
   1:  PR[GP1:91,1] = PR[GP1:90,1] + -39.634;
   1:  PR[GP1:91,2] = PR[GP1:90,2] + 8.697;
   1:L PR[91] R[100]mm/sec CNT100;
   1:  PR[GP1:91,1] = PR[GP1:90,1] + -40.613;
   1:  PR[GP1:91,2] = PR[GP1:90,2] + 6.439;
   1:L PR[91] R[100]mm/sec CNT100;
   1:  PR[GP1:91,1] = PR[GP1:90,1] + -41.007;
   1:  PR[GP1:91,2] = PR[GP1:90,2] + 5.485;
   1:L PR[91] R[100]mm/sec CNT100;
   1:  PR[GP1:91,1] = PR[GP1:90,1] + -41.586;
   1:  PR[GP1:91,2] = PR[GP1:90,2] + 3.175;
   1:L PR[91] R[100]mm/sec CNT100;
   1:  PR[GP1:91,1] = PR[GP1:90,1] + -41.792;
   1:  PR[GP1:91,2] = PR[GP1:90,2] + 0.662;
   1:L PR[91] R[100]mm/sec CNT100;
   1:  PR[GP1:91,1] = PR[GP1:90,1] + -41.923;
   1:  PR[GP1:91,2] = PR[GP1:90,2] + -0.346;
   1:L PR[91] R[100]mm/sec CNT100;
   1:  PR[GP1:91,1] = PR[GP1:90,1] + -41.723;
   1:  PR[GP1:91,2] = PR[GP1:90,2] + -2.779;
   1:L PR[91] R[100]mm/sec CNT100;
   1:  PR[GP1:91,1] = PR[GP1:90,1] + -41.594;
   1:  PR[GP1:91,2] = PR[GP1:90,2] + -3.765;
   1:L PR[91] R[100]mm/sec CNT100;
   1:  PR[GP1:91,1] = PR[GP1:90,1] + -41.010;
   1:  PR[GP1:91,2] = PR[GP1:90,2] + -6.097;
   1:L PR[91] R[100]mm/sec CNT100;
   1:  PR[GP1:91,1] = PR[GP1:90,1] + -40.015;
   1:  PR[GP1:91,2] = PR[GP1:90,2] + -8.391;
   1:L PR[91] R[100]mm/sec CNT100;
   1:  PR[GP1:91,1] = PR[GP1:90,1] + -39.627;
   1:  PR[GP1:91,2] = PR[GP1:90,2] + -9.331;
   1:L PR[91] R[100]mm/sec CNT100;
   1:  PR[GP1:91,1] = PR[GP1:90,1] + -38.324;
   1:  PR[GP1:91,2] = PR[GP1:90,2] + -11.351;
   1:L PR[91] R[100]mm/sec CNT100;
   1:  PR[GP1:91,1] = PR[GP1:90,1] + -37.681;
   1:  PR[GP1:91,2] = PR[GP1:90,2] + -12.194;
   1:L PR[91] R[100]mm/sec CNT100;
   1:  PR[GP1:91,1] = PR[GP1:90,1] + -36.079;
   1:  PR[GP1:91,2] = PR[GP1:90,2] + -13.960;
   1:L PR[91] R[100]mm/sec CNT100;
   1:  PR[GP1:91,1] = PR[GP1:90,1] + -33.297;
   1:  PR[GP1:91,2] = PR[GP1:90,2] + -16.150;
   1:L PR[91] R[100]mm/sec CNT100;
   1:  PR[GP1:91,1] = PR[GP1:90,1] + -31.252;
   1:  PR[GP1:91,2] = PR[GP1:90,2] + -17.285;
   1:L PR[91] R[100]mm/sec CNT100;
   1:  PR[GP1:91,1] = PR[GP1:90,1] + -30.166;
   1:  PR[GP1:91,2] = PR[GP1:90,2] + -17.742;
   1:L PR[91] R[100]mm/sec CNT100;
   1:  PR[GP1:91,1] = PR[GP1:90,1] + -27.972;
   1:  PR[GP1:91,2] = PR[GP1:90,2] + -18.526;
   1:L PR[91] R[100]mm/sec CNT100;
   1:  PR[GP1:91,1] = PR[GP1:90,1] + -25.669;
   1:  PR[GP1:91,2] = PR[GP1:90,2] + -18.944;
   1:L PR[91] R[100]mm/sec CNT100;
   1:  PR[GP1:91,1] = PR[GP1:90,1] + -24.444;
   1:  PR[GP1:91,2] = PR[GP1:90,2] + -19.115;
   1:L PR[91] R[100]mm/sec CNT100;
   1:  PR[GP1:91,1] = PR[GP1:90,1] + -22.218;
   1:  PR[GP1:91,2] = PR[GP1:90,2] + -19.150;
   1:L PR[91] R[100]mm/sec CNT100;
   1:  PR[GP1:91,1] = PR[GP1:90,1] + -19.907;
   1:  PR[GP1:91,2] = PR[GP1:90,2] + -18.806;
   1:L PR[91] R[100]mm/sec CNT100;
   1:  PR[GP1:91,1] = PR[GP1:90,1] + -18.614;
   1:  PR[GP1:91,2] = PR[GP1:90,2] + -18.651;
   1:L PR[91] R[100]mm/sec CNT100;
   1:  PR[GP1:91,1] = PR[GP1:90,1] + -16.536;
   1:  PR[GP1:91,2] = PR[GP1:90,2] + -17.981;
   1:L PR[91] R[100]mm/sec CNT100;
   1:  PR[GP1:91,1] = PR[GP1:90,1] + -15.199;
   1:  PR[GP1:91,2] = PR[GP1:90,2] + -17.447;
   1:L PR[91] R[100]mm/sec CNT100;
   1:  PR[GP1:91,1] = PR[GP1:90,1] + -13.314;
   1:  PR[GP1:91,2] = PR[GP1:90,2] + -16.477;
   1:L PR[91] R[100]mm/sec CNT100;
   1:  PR[GP1:91,1] = PR[GP1:90,1] + -10.340;
   1:  PR[GP1:91,2] = PR[GP1:90,2] + -14.267;
   1:L PR[91] R[100]mm/sec CNT100;
   1:  PR[GP1:91,1] = PR[GP1:90,1] + -8.914;
   1:  PR[GP1:91,2] = PR[GP1:90,2] + -12.791;
   1:L PR[91] R[100]mm/sec CNT100;
   1:  PR[GP1:91,1] = PR[GP1:90,1] + -7.888;
   1:  PR[GP1:91,2] = PR[GP1:90,2] + -11.498;
   1:L PR[91] R[100]mm/sec CNT100;
   1:  PR[GP1:91,1] = PR[GP1:90,1] + -6.741;
   1:  PR[GP1:91,2] = PR[GP1:90,2] + -9.836;
   1:L PR[91] R[100]mm/sec CNT100;
   1:  PR[GP1:91,1] = PR[GP1:90,1] + -5.868;
   1:  PR[GP1:91,2] = PR[GP1:90,2] + -7.985;
   1:L PR[91] R[100]mm/sec CNT100;
   1:  PR[GP1:91,1] = PR[GP1:90,1] + -5.185;
   1:  PR[GP1:91,2] = PR[GP1:90,2] + -6.416;
   1:L PR[91] R[100]mm/sec CNT100;
   1:  PR[GP1:91,1] = PR[GP1:90,1] + -4.813;
   1:  PR[GP1:91,2] = PR[GP1:90,2] + -5.108;
   1:L PR[91] R[100]mm/sec CNT100;
   1:  PR[GP1:91,1] = PR[GP1:90,1] + -4.861;
   1:  PR[GP1:91,2] = PR[GP1:90,2] + -5.039;
   1:L PR[91] R[100]mm/sec CNT100;
   1:  PR[GP1:91,1] = PR[GP1:90,1] + -4.361;
   1:  PR[GP1:91,2] = PR[GP1:90,2] + -3.647;
   1:L PR[91] R[100]mm/sec CNT100;
   1:  PR[GP1:91,1] = PR[GP1:90,1] + -3.618;
   1:  PR[GP1:91,2] = PR[GP1:90,2] + -2.688;
   1:L PR[91] R[100]mm/sec CNT100;
   1:  PR[GP1:91,1] = PR[GP1:90,1] + -2.659;
   1:  PR[GP1:91,2] = PR[GP1:90,2] + -2.075;
   1:L PR[91] R[100]mm/sec CNT100;
   1:  PR[GP1:91,1] = PR[GP1:90,1] + -1.667;
   1:  PR[GP1:91,2] = PR[GP1:90,2] + -1.882;
   1:L PR[91] R[100]mm/sec CNT100;
   1:  PR[GP1:91,1] = PR[GP1:90,1] + 1.823;
   1:L PR[91] R[100]mm/sec CNT100;
   1:  PR[GP1:91,1] = PR[GP1:90,1] + 2.813;
   1:  PR[GP1:91,2] = PR[GP1:90,2] + -2.075;
   1:L PR[91] R[100]mm/sec CNT100;
   1:  PR[GP1:91,1] = PR[GP1:90,1] + 3.550;
   1:  PR[GP1:91,2] = PR[GP1:90,2] + -2.542;
   1:L PR[91] R[100]mm/sec CNT100;
   1:  PR[GP1:91,1] = PR[GP1:90,1] + 3.793;
   1:  PR[GP1:91,2] = PR[GP1:90,2] + -2.711;
   1:L PR[91] R[100]mm/sec CNT100;
   1:  PR[GP1:91,1] = PR[GP1:90,1] + 4.524;
   1:  PR[GP1:91,2] = PR[GP1:90,2] + -3.657;
   1:L PR[91] R[100]mm/sec CNT100;
   1:  PR[GP1:91,1] = PR[GP1:90,1] + 4.785;
   1:  PR[GP1:91,2] = PR[GP1:90,2] + -4.383;
   1:L PR[91] R[100]mm/sec CNT100;
   1:  PR[GP1:91,1] = PR[GP1:90,1] + 5.323;
   1:  PR[GP1:91,2] = PR[GP1:90,2] + -6.332;
   1:L PR[91] R[100]mm/sec CNT100;
   1:  PR[GP1:91,1] = PR[GP1:90,1] + 6.167;
   1:  PR[GP1:91,2] = PR[GP1:90,2] + -8.121;
   1:L PR[91] R[100]mm/sec CNT100;
   1:  PR[GP1:91,1] = PR[GP1:90,1] + 6.911;
   1:  PR[GP1:91,2] = PR[GP1:90,2] + -9.855;
   1:L PR[91] R[100]mm/sec CNT100;
   1:  PR[GP1:91,1] = PR[GP1:90,1] + 8.045;
   1:  PR[GP1:91,2] = PR[GP1:90,2] + -11.496;
   1:L PR[91] R[100]mm/sec CNT100;
   1:  PR[GP1:91,1] = PR[GP1:90,1] + 9.070;
   1:  PR[GP1:91,2] = PR[GP1:90,2] + -12.790;
   1:L PR[91] R[100]mm/sec CNT100;
   1:  PR[GP1:91,1] = PR[GP1:90,1] + 10.497;
   1:  PR[GP1:91,2] = PR[GP1:90,2] + -14.267;
   1:L PR[91] R[100]mm/sec CNT100;
   1:  PR[GP1:91,1] = PR[GP1:90,1] + 13.470;
   1:  PR[GP1:91,2] = PR[GP1:90,2] + -16.477;
   1:L PR[91] R[100]mm/sec CNT100;
   1:  PR[GP1:91,1] = PR[GP1:90,1] + 15.355;
   1:  PR[GP1:91,2] = PR[GP1:90,2] + -17.447;
   1:L PR[91] R[100]mm/sec CNT100;
   1:  PR[GP1:91,1] = PR[GP1:90,1] + 16.692;
   1:  PR[GP1:91,2] = PR[GP1:90,2] + -17.981;
   1:L PR[91] R[100]mm/sec CNT100;
   1:  PR[GP1:91,1] = PR[GP1:90,1] + 18.790;
   1:  PR[GP1:91,2] = PR[GP1:90,2] + -18.657;
   1:L PR[91] R[100]mm/sec CNT100;
   1:  PR[GP1:91,1] = PR[GP1:90,1] + 21.000;
   1:  PR[GP1:91,2] = PR[GP1:90,2] + -18.986;
   1:L PR[91] R[100]mm/sec CNT100;
   1:  PR[GP1:91,1] = PR[GP1:90,1] + 22.354;
   1:  PR[GP1:91,2] = PR[GP1:90,2] + -19.150;
   1:L PR[91] R[100]mm/sec CNT100;
   1:  PR[GP1:91,1] = PR[GP1:90,1] + 24.571;
   1:  PR[GP1:91,2] = PR[GP1:90,2] + -19.115;
   1:L PR[91] R[100]mm/sec CNT100;
   1:  PR[GP1:91,1] = PR[GP1:90,1] + 26.877;
   1:  PR[GP1:91,2] = PR[GP1:90,2] + -18.697;
   1:L PR[91] R[100]mm/sec CNT100;
   1:  PR[GP1:91,1] = PR[GP1:90,1] + 28.155;
   1:  PR[GP1:91,2] = PR[GP1:90,2] + -18.516;
   1:L PR[91] R[100]mm/sec CNT100;
   1:  PR[GP1:91,1] = PR[GP1:90,1] + 30.322;
   1:  PR[GP1:91,2] = PR[GP1:90,2] + -17.742;
   1:L PR[91] R[100]mm/sec CNT100;
   1:  PR[GP1:91,1] = PR[GP1:90,1] + 31.409;
   1:  PR[GP1:91,2] = PR[GP1:90,2] + -17.285;
   1:L PR[91] R[100]mm/sec CNT100;
   1:  PR[GP1:91,1] = PR[GP1:90,1] + 33.453;
   1:  PR[GP1:91,2] = PR[GP1:90,2] + -16.150;
   1:L PR[91] R[100]mm/sec CNT100;
   1:  PR[GP1:91,1] = PR[GP1:90,1] + 36.236;
   1:  PR[GP1:91,2] = PR[GP1:90,2] + -13.960;
   1:L PR[91] R[100]mm/sec CNT100;
   1:  PR[GP1:91,1] = PR[GP1:90,1] + 37.838;
   1:  PR[GP1:91,2] = PR[GP1:90,2] + -12.194;
   1:L PR[91] R[100]mm/sec CNT100;
   1:  PR[GP1:91,1] = PR[GP1:90,1] + 38.481;
   1:  PR[GP1:91,2] = PR[GP1:90,2] + -11.351;
   1:L PR[91] R[100]mm/sec CNT100;
   1:  PR[GP1:91,1] = PR[GP1:90,1] + 39.791;
   1:  PR[GP1:91,2] = PR[GP1:90,2] + -9.320;
   1:L PR[91] R[100]mm/sec CNT100;
   1:  PR[GP1:91,1] = PR[GP1:90,1] + 40.770;
   1:  PR[GP1:91,2] = PR[GP1:90,2] + -7.063;
   1:L PR[91] R[100]mm/sec CNT100;
   1:  PR[GP1:91,1] = PR[GP1:90,1] + 41.164;
   1:  PR[GP1:91,2] = PR[GP1:90,2] + -6.110;
   1:L PR[91] R[100]mm/sec CNT100;
   1:  PR[GP1:91,1] = PR[GP1:90,1] + 41.743;
   1:  PR[GP1:91,2] = PR[GP1:90,2] + -3.800;
   1:L PR[91] R[100]mm/sec CNT100;
   1:  PR[GP1:91,1] = PR[GP1:90,1] + 41.949;
   1:  PR[GP1:91,2] = PR[GP1:90,2] + -1.287;
   1:L PR[91] R[100]mm/sec CNT100;
   1:  PR[GP1:91,1] = PR[GP1:90,1] + 42.080;
   1:  PR[GP1:91,2] = PR[GP1:90,2] + -0.278;
   1:L PR[91] R[100]mm/sec CNT100;
   1:  PR[GP1:91,1] = PR[GP1:90,1] + 41.880;
   1:  PR[GP1:91,2] = PR[GP1:90,2] + 2.155;
   1:L PR[91] R[100]mm/sec CNT100;
   1:  PR[GP1:91,1] = PR[GP1:90,1] + 41.751;
   1:  PR[GP1:91,2] = PR[GP1:90,2] + 3.142;
   1:L PR[91] R[100]mm/sec CNT100;
   1:  PR[GP1:91,1] = PR[GP1:90,1] + 41.167;
   1:  PR[GP1:91,2] = PR[GP1:90,2] + 5.474;
   1:L PR[91] R[100]mm/sec CNT100;
   1:  PR[GP1:91,1] = PR[GP1:90,1] + 40.172;
   1:  PR[GP1:91,2] = PR[GP1:90,2] + 7.767;
   1:L PR[91] R[100]mm/sec CNT100;
   1:  PR[GP1:91,1] = PR[GP1:90,1] + 39.784;
   1:  PR[GP1:91,2] = PR[GP1:90,2] + 8.707;
   1:L PR[91] R[100]mm/sec CNT100;
   1:  PR[GP1:91,1] = PR[GP1:90,1] + 38.481;
   1:  PR[GP1:91,2] = PR[GP1:90,2] + 10.727;
   1:L PR[91] R[100]mm/sec CNT100;
   1:  PR[GP1:91,1] = PR[GP1:90,1] + 37.837;
   1:  PR[GP1:91,2] = PR[GP1:90,2] + 11.570;
   1:L PR[91] R[100]mm/sec CNT100;
   1:  PR[GP1:91,1] = PR[GP1:90,1] + 36.236;
   1:  PR[GP1:91,2] = PR[GP1:90,2] + 13.337;
   1:L PR[91] R[100]mm/sec CNT100;
   1:  PR[GP1:91,1] = PR[GP1:90,1] + 33.452;
   1:  PR[GP1:91,2] = PR[GP1:90,2] + 15.526;
   1:L PR[91] R[100]mm/sec CNT100;
   1:  PR[GP1:91,1] = PR[GP1:90,1] + 31.408;
   1:  PR[GP1:91,2] = PR[GP1:90,2] + 16.661;
   1:L PR[91] R[100]mm/sec CNT100;
   1:  PR[GP1:91,1] = PR[GP1:90,1] + 30.321;
   1:  PR[GP1:91,2] = PR[GP1:90,2] + 17.119;
   1:L PR[91] R[100]mm/sec CNT100;
   1:  PR[GP1:91,1] = PR[GP1:90,1] + 28.127;
   1:  PR[GP1:91,2] = PR[GP1:90,2] + 17.902;
   1:L PR[91] R[100]mm/sec CNT100;
   1:  PR[GP1:91,1] = PR[GP1:90,1] + 25.825;
   1:  PR[GP1:91,2] = PR[GP1:90,2] + 18.320;
   1:L PR[91] R[100]mm/sec CNT100;
   1:  PR[GP1:91,1] = PR[GP1:90,1] + 24.599;
   1:  PR[GP1:91,2] = PR[GP1:90,2] + 18.491;
   1:L PR[91] R[100]mm/sec CNT100;
   1:  PR[GP1:91,1] = PR[GP1:90,1] + 22.372;
   1:  PR[GP1:91,2] = PR[GP1:90,2] + 18.526;
   1:L PR[91] R[100]mm/sec CNT100;
   1:  PR[GP1:91,1] = PR[GP1:90,1] + 20.062;
   1:  PR[GP1:91,2] = PR[GP1:90,2] + 18.182;
   1:L PR[91] R[100]mm/sec CNT100;
   1:  PR[GP1:91,1] = PR[GP1:90,1] + 18.769;
   1:  PR[GP1:91,2] = PR[GP1:90,2] + 18.026;
   1:L PR[91] R[100]mm/sec CNT100;
   1:  PR[GP1:91,1] = PR[GP1:90,1] + 16.690;
   1:  PR[GP1:91,2] = PR[GP1:90,2] + 17.357;
   1:L PR[91] R[100]mm/sec CNT100;
   1:  PR[GP1:91,1] = PR[GP1:90,1] + 15.353;
   1:  PR[GP1:91,2] = PR[GP1:90,2] + 16.821;
   1:L PR[91] R[100]mm/sec CNT100;
   1:  PR[GP1:91,1] = PR[GP1:90,1] + 13.468;
   1:  PR[GP1:91,2] = PR[GP1:90,2] + 15.851;
   1:L PR[91] R[100]mm/sec CNT100;
   1:  PR[GP1:91,1] = PR[GP1:90,1] + 10.494;
   1:  PR[GP1:91,2] = PR[GP1:90,2] + 13.641;
   1:L PR[91] R[100]mm/sec CNT100;
   1:  PR[GP1:91,1] = PR[GP1:90,1] + 9.068;
   1:  PR[GP1:91,2] = PR[GP1:90,2] + 12.164;
   1:L PR[91] R[100]mm/sec CNT100;
   1:  PR[GP1:91,1] = PR[GP1:90,1] + 8.043;
   1:  PR[GP1:91,2] = PR[GP1:90,2] + 10.869;
   1:L PR[91] R[100]mm/sec CNT100;
   1:  PR[GP1:91,1] = PR[GP1:90,1] + 6.895;
   1:  PR[GP1:91,2] = PR[GP1:90,2] + 9.207;
   1:L PR[91] R[100]mm/sec CNT100;
   1:  PR[GP1:91,1] = PR[GP1:90,1] + 6.021;
   1:  PR[GP1:91,2] = PR[GP1:90,2] + 7.354;
   1:L PR[91] R[100]mm/sec CNT100;
   1:  PR[GP1:91,1] = PR[GP1:90,1] + 5.347;
   1:  PR[GP1:91,2] = PR[GP1:90,2] + 5.821;
   1:L PR[91] R[100]mm/sec CNT100;
   1:  PR[GP1:91,1] = PR[GP1:90,1] + 4.972;
   1:  PR[GP1:91,2] = PR[GP1:90,2] + 4.499;
   1:L PR[91] R[100]mm/sec CNT100;
   1:  PR[GP1:91,1] = PR[GP1:90,1] + 5.022;
   1:  PR[GP1:91,2] = PR[GP1:90,2] + 4.431;
   1:L PR[91] R[100]mm/sec CNT100;
   1:  PR[GP1:91,1] = PR[GP1:90,1] + 4.515;
   1:  PR[GP1:91,2] = PR[GP1:90,2] + 3.018;
   1:L PR[91] R[100]mm/sec CNT100;
   1:  PR[GP1:91,1] = PR[GP1:90,1] + 3.793;
   1:  PR[GP1:91,2] = PR[GP1:90,2] + 2.087;
   1:L PR[91] R[100]mm/sec CNT100;
   1:  PR[GP1:91,1] = PR[GP1:90,1] + 3.551;
   1:  PR[GP1:91,2] = PR[GP1:90,2] + 1.919;
   1:L PR[91] R[100]mm/sec CNT100;
   1:  PR[GP1:91,1] = PR[GP1:90,1] + 2.813;
   1:  PR[GP1:91,2] = PR[GP1:90,2] + 1.451;
   1:L PR[91] R[100]mm/sec CNT100;
   1:  PR[GP1:91,1] = PR[GP1:90,1] + 1.823;
   1:  PR[GP1:91,2] = PR[GP1:90,2] + 1.258;
   1:L PR[91] R[100]mm/sec CNT100;
   1:  PR[GP1:91,1] = PR[GP1:90,1] + -1.668;
   1:L PR[91] R[100]mm/sec CNT100;
   1:  PR[91] = PR[90];
   1:  PR[GP1:91,1] = PR[GP1:90,1] + -2.657;
   1:  PR[GP1:91,2] = PR[GP1:90,2] + 1.743;
   1:  PR[GP1:91,3] = PR[GP1:90,3] + 7.015;
   1:L PR[91] R[100]mm/sec CNT100;
   1:  PR[GP1:91,1] = PR[GP1:90,1] + -3.626;
   1:  PR[GP1:91,2] = PR[GP1:90,2] + 2.366;
   1:L PR[91] R[100]mm/sec CNT100;
   1:  PR[GP1:91,1] = PR[GP1:90,1] + -4.139;
   1:  PR[GP1:91,2] = PR[GP1:90,2] + 3.050;
   1:L PR[91] R[100]mm/sec CNT100;
   1:  PR[GP1:91,1] = PR[GP1:90,1] + -4.410;
   1:  PR[GP1:91,2] = PR[GP1:90,2] + 3.366;
   1:L PR[91] R[100]mm/sec CNT100;
   1:  PR[GP1:91,1] = PR[GP1:90,1] + -4.642;
   1:  PR[GP1:91,2] = PR[GP1:90,2] + 4.008;
   1:L PR[91] R[100]mm/sec CNT100;
   1:  PR[GP1:91,1] = PR[GP1:90,1] + -5.034;
   1:  PR[GP1:91,2] = PR[GP1:90,2] + 5.430;
   1:L PR[91] R[100]mm/sec CNT100;
   1:  PR[GP1:91,1] = PR[GP1:90,1] + -5.646;
   1:  PR[GP1:91,2] = PR[GP1:90,2] + 6.729;
   1:L PR[91] R[100]mm/sec CNT100;
   1:  PR[GP1:91,1] = PR[GP1:90,1] + -6.738;
   1:  PR[GP1:91,2] = PR[GP1:90,2] + 9.280;
   1:L PR[91] R[100]mm/sec CNT100;
   1:  PR[GP1:91,1] = PR[GP1:90,1] + -7.601;
   1:  PR[GP1:91,2] = PR[GP1:90,2] + 10.531;
   1:L PR[91] R[100]mm/sec CNT100;
   1:  PR[GP1:91,1] = PR[GP1:90,1] + -9.086;
   1:  PR[GP1:91,2] = PR[GP1:90,2] + 12.403;
   1:L PR[91] R[100]mm/sec CNT100;
   1:  PR[GP1:91,1] = PR[GP1:90,1] + -10.200;
   1:  PR[GP1:91,2] = PR[GP1:90,2] + 13.556;
   1:L PR[91] R[100]mm/sec CNT100;
   1:  PR[GP1:91,1] = PR[GP1:90,1] + -13.382;
   1:  PR[GP1:91,2] = PR[GP1:90,2] + 15.920;
   1:L PR[91] R[100]mm/sec CNT100;
   1:  PR[GP1:91,1] = PR[GP1:90,1] + -14.890;
   1:  PR[GP1:91,2] = PR[GP1:90,2] + 16.696;
   1:L PR[91] R[100]mm/sec CNT100;
   1:  PR[GP1:91,1] = PR[GP1:90,1] + -16.831;
   1:  PR[GP1:91,2] = PR[GP1:90,2] + 17.473;
   1:L PR[91] R[100]mm/sec CNT100;
   1:  PR[GP1:91,1] = PR[GP1:90,1] + -18.553;
   1:  PR[GP1:91,2] = PR[GP1:90,2] + 18.027;
   1:L PR[91] R[100]mm/sec CNT100;
   1:  PR[GP1:91,1] = PR[GP1:90,1] + -20.372;
   1:  PR[GP1:91,2] = PR[GP1:90,2] + 18.298;
   1:L PR[91] R[100]mm/sec CNT100;
   1:  PR[GP1:91,1] = PR[GP1:90,1] + -22.340;
   1:  PR[GP1:91,2] = PR[GP1:90,2] + 18.536;
   1:L PR[91] R[100]mm/sec CNT100;
   1:  PR[GP1:91,1] = PR[GP1:90,1] + -24.188;
   1:  PR[GP1:91,2] = PR[GP1:90,2] + 18.507;
   1:L PR[91] R[100]mm/sec CNT100;
   1:  PR[GP1:91,1] = PR[GP1:90,1] + -26.130;
   1:  PR[GP1:91,2] = PR[GP1:90,2] + 18.155;
   1:L PR[91] R[100]mm/sec CNT100;
   1:  PR[GP1:91,1] = PR[GP1:90,1] + -27.990;
   1:  PR[GP1:91,2] = PR[GP1:90,2] + 17.892;
   1:L PR[91] R[100]mm/sec CNT100;
   1:  PR[GP1:91,1] = PR[GP1:90,1] + -29.830;
   1:  PR[GP1:91,2] = PR[GP1:90,2] + 17.235;
   1:L PR[91] R[100]mm/sec CNT100;
   1:  PR[GP1:91,1] = PR[GP1:90,1] + -31.416;
   1:  PR[GP1:91,2] = PR[GP1:90,2] + 16.567;
   1:L PR[91] R[100]mm/sec CNT100;
   1:  PR[GP1:91,1] = PR[GP1:90,1] + -33.170;
   1:  PR[GP1:91,2] = PR[GP1:90,2] + 15.593;
   1:L PR[91] R[100]mm/sec CNT100;
   1:  PR[GP1:91,1] = PR[GP1:90,1] + -34.811;
   1:  PR[GP1:91,2] = PR[GP1:90,2] + 14.292;
   1:L PR[91] R[100]mm/sec CNT100;
   1:  PR[GP1:91,1] = PR[GP1:90,1] + -36.113;
   1:  PR[GP1:91,2] = PR[GP1:90,2] + 13.283;
   1:L PR[91] R[100]mm/sec CNT100;
   1:  PR[GP1:91,1] = PR[GP1:90,1] + -37.500;
   1:  PR[GP1:91,2] = PR[GP1:90,2] + 11.754;
   1:L PR[91] R[100]mm/sec CNT100;
   1:  PR[GP1:91,1] = PR[GP1:90,1] + -38.441;
   1:  PR[GP1:91,2] = PR[GP1:90,2] + 10.520;
   1:L PR[91] R[100]mm/sec CNT100;
   1:  PR[GP1:91,1] = PR[GP1:90,1] + -39.586;
   1:  PR[GP1:91,2] = PR[GP1:90,2] + 8.745;
   1:L PR[91] R[100]mm/sec CNT100;
   1:  PR[GP1:91,1] = PR[GP1:90,1] + -40.444;
   1:  PR[GP1:91,2] = PR[GP1:90,2] + 6.767;
   1:L PR[91] R[100]mm/sec CNT100;
   1:  PR[GP1:91,1] = PR[GP1:90,1] + -41.021;
   1:  PR[GP1:91,2] = PR[GP1:90,2] + 5.369;
   1:L PR[91] R[100]mm/sec CNT100;
   1:  PR[GP1:91,1] = PR[GP1:90,1] + -41.528;
   1:  PR[GP1:91,2] = PR[GP1:90,2] + 3.348;
   1:L PR[91] R[100]mm/sec CNT100;
   1:  PR[GP1:91,1] = PR[GP1:90,1] + -41.710;
   1:  PR[GP1:91,2] = PR[GP1:90,2] + 1.133;
   1:L PR[91] R[100]mm/sec CNT100;
   1:  PR[GP1:91,1] = PR[GP1:90,1] + -41.901;
   1:  PR[GP1:91,2] = PR[GP1:90,2] + -0.346;
   1:L PR[91] R[100]mm/sec CNT100;
   1:  PR[GP1:91,1] = PR[GP1:90,1] + -41.726;
   1:  PR[GP1:91,2] = PR[GP1:90,2] + -2.491;
   1:L PR[91] R[100]mm/sec CNT100;
   1:  PR[GP1:91,1] = PR[GP1:90,1] + -41.536;
   1:  PR[GP1:91,2] = PR[GP1:90,2] + -3.938;
   1:L PR[91] R[100]mm/sec CNT100;
   1:  PR[GP1:91,1] = PR[GP1:90,1] + -41.025;
   1:  PR[GP1:91,2] = PR[GP1:90,2] + -5.981;
   1:L PR[91] R[100]mm/sec CNT100;
   1:  PR[GP1:91,1] = PR[GP1:90,1] + -40.148;
   1:  PR[GP1:91,2] = PR[GP1:90,2] + -8.001;
   1:L PR[91] R[100]mm/sec CNT100;
   1:  PR[GP1:91,1] = PR[GP1:90,1] + -39.579;
   1:  PR[GP1:91,2] = PR[GP1:90,2] + -9.380;
   1:L PR[91] R[100]mm/sec CNT100;
   1:  PR[GP1:91,1] = PR[GP1:90,1] + -38.441;
   1:  PR[GP1:91,2] = PR[GP1:90,2] + -11.144;
   1:L PR[91] R[100]mm/sec CNT100;
   1:  PR[GP1:91,1] = PR[GP1:90,1] + -37.500;
   1:  PR[GP1:91,2] = PR[GP1:90,2] + -12.378;
   1:L PR[91] R[100]mm/sec CNT100;
   1:  PR[GP1:91,1] = PR[GP1:90,1] + -36.107;
   1:  PR[GP1:91,2] = PR[GP1:90,2] + -13.914;
   1:L PR[91] R[100]mm/sec CNT100;
   1:  PR[GP1:91,1] = PR[GP1:90,1] + -34.442;
   1:  PR[GP1:91,2] = PR[GP1:90,2] + -15.234;
   1:L PR[91] R[100]mm/sec CNT100;
   1:  PR[GP1:91,1] = PR[GP1:90,1] + -33.178;
   1:  PR[GP1:91,2] = PR[GP1:90,2] + -16.213;
   1:L PR[91] R[100]mm/sec CNT100;
   1:  PR[GP1:91,1] = PR[GP1:90,1] + -31.416;
   1:  PR[GP1:91,2] = PR[GP1:90,2] + -17.191;
   1:L PR[91] R[100]mm/sec CNT100;
   1:  PR[GP1:91,1] = PR[GP1:90,1] + -29.830;
   1:  PR[GP1:91,2] = PR[GP1:90,2] + -17.859;
   1:L PR[91] R[100]mm/sec CNT100;
   1:  PR[GP1:91,1] = PR[GP1:90,1] + -27.964;
   1:  PR[GP1:91,2] = PR[GP1:90,2] + -18.525;
   1:L PR[91] R[100]mm/sec CNT100;
   1:  PR[GP1:91,1] = PR[GP1:90,1] + -26.003;
   1:  PR[GP1:91,2] = PR[GP1:90,2] + -18.881;
   1:L PR[91] R[100]mm/sec CNT100;
   1:  PR[GP1:91,1] = PR[GP1:90,1] + -24.217;
   1:  PR[GP1:91,2] = PR[GP1:90,2] + -19.131;
   1:L PR[91] R[100]mm/sec CNT100;
   1:  PR[GP1:91,1] = PR[GP1:90,1] + -22.360;
   1:  PR[GP1:91,2] = PR[GP1:90,2] + -19.160;
   1:L PR[91] R[100]mm/sec CNT100;
   1:  PR[GP1:91,1] = PR[GP1:90,1] + -20.415;
   1:  PR[GP1:91,2] = PR[GP1:90,2] + -18.870;
   1:L PR[91] R[100]mm/sec CNT100;
   1:  PR[GP1:91,1] = PR[GP1:90,1] + -18.534;
   1:  PR[GP1:91,2] = PR[GP1:90,2] + -18.645;
   1:L PR[91] R[100]mm/sec CNT100;
   1:  PR[GP1:91,1] = PR[GP1:90,1] + -16.832;
   1:  PR[GP1:91,2] = PR[GP1:90,2] + -18.097;
   1:L PR[91] R[100]mm/sec CNT100;
   1:  PR[GP1:91,1] = PR[GP1:90,1] + -14.891;
   1:  PR[GP1:91,2] = PR[GP1:90,2] + -17.321;
   1:L PR[91] R[100]mm/sec CNT100;
   1:  PR[GP1:91,1] = PR[GP1:90,1] + -13.382;
   1:  PR[GP1:91,2] = PR[GP1:90,2] + -16.544;
   1:L PR[91] R[100]mm/sec CNT100;
   1:  PR[GP1:91,1] = PR[GP1:90,1] + -10.200;
   1:  PR[GP1:91,2] = PR[GP1:90,2] + -14.180;
   1:L PR[91] R[100]mm/sec CNT100;
   1:  PR[GP1:91,1] = PR[GP1:90,1] + -9.086;
   1:  PR[GP1:91,2] = PR[GP1:90,2] + -13.027;
   1:L PR[91] R[100]mm/sec CNT100;
   1:  PR[GP1:91,1] = PR[GP1:90,1] + -7.602;
   1:  PR[GP1:91,2] = PR[GP1:90,2] + -11.155;
   1:L PR[91] R[100]mm/sec CNT100;
   1:  PR[GP1:91,1] = PR[GP1:90,1] + -6.723;
   1:  PR[GP1:91,2] = PR[GP1:90,2] + -9.883;
   1:L PR[91] R[100]mm/sec CNT100;
   1:  PR[GP1:91,1] = PR[GP1:90,1] + -6.052;
   1:  PR[GP1:91,2] = PR[GP1:90,2] + -8.461;
   1:L PR[91] R[100]mm/sec CNT100;
   1:  PR[GP1:91,1] = PR[GP1:90,1] + -5.064;
   1:  PR[GP1:91,2] = PR[GP1:90,2] + -6.190;
   1:L PR[91] R[100]mm/sec CNT100;
   1:  PR[GP1:91,1] = PR[GP1:90,1] + -4.826;
   1:  PR[GP1:91,2] = PR[GP1:90,2] + -5.354;
   1:L PR[91] R[100]mm/sec CNT100;
   1:  PR[GP1:91,1] = PR[GP1:90,1] + -4.872;
   1:  PR[GP1:91,2] = PR[GP1:90,2] + -5.290;
   1:L PR[91] R[100]mm/sec CNT100;
   1:  PR[GP1:91,1] = PR[GP1:90,1] + -4.392;
   1:  PR[GP1:91,2] = PR[GP1:90,2] + -3.953;
   1:L PR[91] R[100]mm/sec CNT100;
   1:  PR[GP1:91,1] = PR[GP1:90,1] + -4.128;
   1:  PR[GP1:91,2] = PR[GP1:90,2] + -3.661;
   1:L PR[91] R[100]mm/sec CNT100;
   1:  PR[GP1:91,1] = PR[GP1:90,1] + -3.626;
   1:  PR[GP1:91,2] = PR[GP1:90,2] + -2.990;
   1:L PR[91] R[100]mm/sec CNT100;
   1:  PR[GP1:91,1] = PR[GP1:90,1] + -2.657;
   1:  PR[GP1:91,2] = PR[GP1:90,2] + -2.367;
   1:L PR[91] R[100]mm/sec CNT100;
   1:  PR[GP1:91,1] = PR[GP1:90,1] + -1.661;
   1:  PR[GP1:91,2] = PR[GP1:90,2] + -2.171;
   1:L PR[91] R[100]mm/sec CNT100;
   1:  PR[GP1:91,1] = PR[GP1:90,1] + 1.816;
   1:L PR[91] R[100]mm/sec CNT100;
   1:  PR[GP1:91,1] = PR[GP1:90,1] + 2.808;
   1:  PR[GP1:91,2] = PR[GP1:90,2] + -2.365;
   1:L PR[91] R[100]mm/sec CNT100;
   1:  PR[GP1:91,1] = PR[GP1:90,1] + 3.505;
   1:  PR[GP1:91,2] = PR[GP1:90,2] + -2.807;
   1:L PR[91] R[100]mm/sec CNT100;
   1:  PR[GP1:91,1] = PR[GP1:90,1] + 3.798;
   1:  PR[GP1:91,2] = PR[GP1:90,2] + -3.011;
   1:L PR[91] R[100]mm/sec CNT100;
   1:  PR[GP1:91,1] = PR[GP1:90,1] + 4.293;
   1:  PR[GP1:91,2] = PR[GP1:90,2] + -3.671;
   1:L PR[91] R[100]mm/sec CNT100;
   1:  PR[GP1:91,1] = PR[GP1:90,1] + 4.563;
   1:  PR[GP1:91,2] = PR[GP1:90,2] + -3.982;
   1:L PR[91] R[100]mm/sec CNT100;
   1:  PR[GP1:91,1] = PR[GP1:90,1] + 4.797;
   1:  PR[GP1:91,2] = PR[GP1:90,2] + -4.633;
   1:L PR[91] R[100]mm/sec CNT100;
   1:  PR[GP1:91,1] = PR[GP1:90,1] + 5.196;
   1:  PR[GP1:91,2] = PR[GP1:90,2] + -6.078;
   1:L PR[91] R[100]mm/sec CNT100;
   1:  PR[GP1:91,1] = PR[GP1:90,1] + 5.818;
   1:  PR[GP1:91,2] = PR[GP1:90,2] + -7.398;
   1:L PR[91] R[100]mm/sec CNT100;
   1:  PR[GP1:91,1] = PR[GP1:90,1] + 6.894;
   1:  PR[GP1:91,2] = PR[GP1:90,2] + -9.902;
   1:L PR[91] R[100]mm/sec CNT100;
   1:  PR[GP1:91,1] = PR[GP1:90,1] + 7.758;
   1:  PR[GP1:91,2] = PR[GP1:90,2] + -11.153;
   1:L PR[91] R[100]mm/sec CNT100;
   1:  PR[GP1:91,1] = PR[GP1:90,1] + 9.242;
   1:  PR[GP1:91,2] = PR[GP1:90,2] + -13.026;
   1:L PR[91] R[100]mm/sec CNT100;
   1:  PR[GP1:91,1] = PR[GP1:90,1] + 10.356;
   1:  PR[GP1:91,2] = PR[GP1:90,2] + -14.179;
   1:L PR[91] R[100]mm/sec CNT100;
   1:  PR[GP1:91,1] = PR[GP1:90,1] + 13.538;
   1:  PR[GP1:91,2] = PR[GP1:90,2] + -16.544;
   1:L PR[91] R[100]mm/sec CNT100;
   1:  PR[GP1:91,1] = PR[GP1:90,1] + 15.047;
   1:  PR[GP1:91,2] = PR[GP1:90,2] + -17.320;
   1:L PR[91] R[100]mm/sec CNT100;
   1:  PR[GP1:91,1] = PR[GP1:90,1] + 16.988;
   1:  PR[GP1:91,2] = PR[GP1:90,2] + -18.096;
   1:L PR[91] R[100]mm/sec CNT100;
   1:  PR[GP1:91,1] = PR[GP1:90,1] + 18.710;
   1:  PR[GP1:91,2] = PR[GP1:90,2] + -18.651;
   1:L PR[91] R[100]mm/sec CNT100;
   1:  PR[GP1:91,1] = PR[GP1:90,1] + 20.528;
   1:  PR[GP1:91,2] = PR[GP1:90,2] + -18.922;
   1:L PR[91] R[100]mm/sec CNT100;
   1:  PR[GP1:91,1] = PR[GP1:90,1] + 22.497;
   1:  PR[GP1:91,2] = PR[GP1:90,2] + -19.160;
   1:L PR[91] R[100]mm/sec CNT100;
   1:  PR[GP1:91,1] = PR[GP1:90,1] + 24.344;
   1:  PR[GP1:91,2] = PR[GP1:90,2] + -19.131;
   1:L PR[91] R[100]mm/sec CNT100;
   1:  PR[GP1:91,1] = PR[GP1:90,1] + 26.286;
   1:  PR[GP1:91,2] = PR[GP1:90,2] + -18.779;
   1:L PR[91] R[100]mm/sec CNT100;
   1:  PR[GP1:91,1] = PR[GP1:90,1] + 28.147;
   1:  PR[GP1:91,2] = PR[GP1:90,2] + -18.516;
   1:L PR[91] R[100]mm/sec CNT100;
   1:  PR[GP1:91,1] = PR[GP1:90,1] + 29.987;
   1:  PR[GP1:91,2] = PR[GP1:90,2] + -17.859;
   1:L PR[91] R[100]mm/sec CNT100;
   1:  PR[GP1:91,1] = PR[GP1:90,1] + 31.572;
   1:  PR[GP1:91,2] = PR[GP1:90,2] + -17.191;
   1:L PR[91] R[100]mm/sec CNT100;
   1:  PR[GP1:91,1] = PR[GP1:90,1] + 33.327;
   1:  PR[GP1:91,2] = PR[GP1:90,2] + -16.217;
   1:L PR[91] R[100]mm/sec CNT100;
   1:  PR[GP1:91,1] = PR[GP1:90,1] + 34.967;
   1:  PR[GP1:91,2] = PR[GP1:90,2] + -14.916;
   1:L PR[91] R[100]mm/sec CNT100;
   1:  PR[GP1:91,1] = PR[GP1:90,1] + 36.270;
   1:  PR[GP1:91,2] = PR[GP1:90,2] + -13.908;
   1:L PR[91] R[100]mm/sec CNT100;
   1:  PR[GP1:91,1] = PR[GP1:90,1] + 37.656;
   1:  PR[GP1:91,2] = PR[GP1:90,2] + -12.379;
   1:L PR[91] R[100]mm/sec CNT100;
   1:  PR[GP1:91,1] = PR[GP1:90,1] + 38.598;
   1:  PR[GP1:91,2] = PR[GP1:90,2] + -11.144;
   1:L PR[91] R[100]mm/sec CNT100;
   1:  PR[GP1:91,1] = PR[GP1:90,1] + 39.743;
   1:  PR[GP1:91,2] = PR[GP1:90,2] + -9.369;
   1:L PR[91] R[100]mm/sec CNT100;
   1:  PR[GP1:91,1] = PR[GP1:90,1] + 40.601;
   1:  PR[GP1:91,2] = PR[GP1:90,2] + -7.391;
   1:L PR[91] R[100]mm/sec CNT100;
   1:  PR[GP1:91,1] = PR[GP1:90,1] + 41.178;
   1:  PR[GP1:91,2] = PR[GP1:90,2] + -5.994;
   1:L PR[91] R[100]mm/sec CNT100;
   1:  PR[GP1:91,1] = PR[GP1:90,1] + 41.685;
   1:  PR[GP1:91,2] = PR[GP1:90,2] + -3.973;
   1:L PR[91] R[100]mm/sec CNT100;
   1:  PR[GP1:91,1] = PR[GP1:90,1] + 41.866;
   1:  PR[GP1:91,2] = PR[GP1:90,2] + -1.758;
   1:L PR[91] R[100]mm/sec CNT100;
   1:  PR[GP1:91,1] = PR[GP1:90,1] + 42.058;
   1:  PR[GP1:91,2] = PR[GP1:90,2] + -0.278;
   1:L PR[91] R[100]mm/sec CNT100;
   1:  PR[GP1:91,1] = PR[GP1:90,1] + 41.882;
   1:  PR[GP1:91,2] = PR[GP1:90,2] + 1.867;
   1:L PR[91] R[100]mm/sec CNT100;
   1:  PR[GP1:91,1] = PR[GP1:90,1] + 41.693;
   1:  PR[GP1:91,2] = PR[GP1:90,2] + 3.316;
   1:L PR[91] R[100]mm/sec CNT100;
   1:  PR[GP1:91,1] = PR[GP1:90,1] + 41.181;
   1:  PR[GP1:91,2] = PR[GP1:90,2] + 5.358;
   1:L PR[91] R[100]mm/sec CNT100;
   1:  PR[GP1:91,1] = PR[GP1:90,1] + 40.305;
   1:  PR[GP1:91,2] = PR[GP1:90,2] + 7.378;
   1:L PR[91] R[100]mm/sec CNT100;
   1:  PR[GP1:91,1] = PR[GP1:90,1] + 39.736;
   1:  PR[GP1:91,2] = PR[GP1:90,2] + 8.756;
   1:L PR[91] R[100]mm/sec CNT100;
   1:  PR[GP1:91,1] = PR[GP1:90,1] + 38.598;
   1:  PR[GP1:91,2] = PR[GP1:90,2] + 10.520;
   1:L PR[91] R[100]mm/sec CNT100;
   1:  PR[GP1:91,1] = PR[GP1:90,1] + 37.656;
   1:  PR[GP1:91,2] = PR[GP1:90,2] + 11.755;
   1:L PR[91] R[100]mm/sec CNT100;
   1:  PR[GP1:91,1] = PR[GP1:90,1] + 36.263;
   1:  PR[GP1:91,2] = PR[GP1:90,2] + 13.291;
   1:L PR[91] R[100]mm/sec CNT100;
   1:  PR[GP1:91,1] = PR[GP1:90,1] + 34.598;
   1:  PR[GP1:91,2] = PR[GP1:90,2] + 14.611;
   1:L PR[91] R[100]mm/sec CNT100;
   1:  PR[GP1:91,1] = PR[GP1:90,1] + 33.333;
   1:  PR[GP1:91,2] = PR[GP1:90,2] + 15.590;
   1:L PR[91] R[100]mm/sec CNT100;
   1:  PR[GP1:91,1] = PR[GP1:90,1] + 31.571;
   1:  PR[GP1:91,2] = PR[GP1:90,2] + 16.568;
   1:L PR[91] R[100]mm/sec CNT100;
   1:  PR[GP1:91,1] = PR[GP1:90,1] + 29.985;
   1:  PR[GP1:91,2] = PR[GP1:90,2] + 17.235;
   1:L PR[91] R[100]mm/sec CNT100;
   1:  PR[GP1:91,1] = PR[GP1:90,1] + 28.118;
   1:  PR[GP1:91,2] = PR[GP1:90,2] + 17.902;
   1:L PR[91] R[100]mm/sec CNT100;
   1:  PR[GP1:91,1] = PR[GP1:90,1] + 26.158;
   1:  PR[GP1:91,2] = PR[GP1:90,2] + 18.258;
   1:L PR[91] R[100]mm/sec CNT100;
   1:  PR[GP1:91,1] = PR[GP1:90,1] + 24.371;
   1:  PR[GP1:91,2] = PR[GP1:90,2] + 18.507;
   1:L PR[91] R[100]mm/sec CNT100;
   1:  PR[GP1:91,1] = PR[GP1:90,1] + 22.514;
   1:  PR[GP1:91,2] = PR[GP1:90,2] + 18.536;
   1:L PR[91] R[100]mm/sec CNT100;
   1:  PR[GP1:91,1] = PR[GP1:90,1] + 20.570;
   1:  PR[GP1:91,2] = PR[GP1:90,2] + 18.246;
   1:L PR[91] R[100]mm/sec CNT100;
   1:  PR[GP1:91,1] = PR[GP1:90,1] + 18.687;
   1:  PR[GP1:91,2] = PR[GP1:90,2] + 18.020;
   1:L PR[91] R[100]mm/sec CNT100;
   1:  PR[GP1:91,1] = PR[GP1:90,1] + 16.985;
   1:  PR[GP1:91,2] = PR[GP1:90,2] + 17.472;
   1:L PR[91] R[100]mm/sec CNT100;
   1:  PR[GP1:91,1] = PR[GP1:90,1] + 15.043;
   1:  PR[GP1:91,2] = PR[GP1:90,2] + 16.694;
   1:L PR[91] R[100]mm/sec CNT100;
   1:  PR[GP1:91,1] = PR[GP1:90,1] + 13.535;
   1:  PR[GP1:91,2] = PR[GP1:90,2] + 15.918;
   1:L PR[91] R[100]mm/sec CNT100;
   1:  PR[GP1:91,1] = PR[GP1:90,1] + 10.352;
   1:  PR[GP1:91,2] = PR[GP1:90,2] + 13.552;
   1:L PR[91] R[100]mm/sec CNT100;
   1:  PR[GP1:91,1] = PR[GP1:90,1] + 9.239;
   1:  PR[GP1:91,2] = PR[GP1:90,2] + 12.399;
   1:L PR[91] R[100]mm/sec CNT100;
   1:  PR[GP1:91,1] = PR[GP1:90,1] + 7.755;
   1:  PR[GP1:91,2] = PR[GP1:90,2] + 10.525;
   1:L PR[91] R[100]mm/sec CNT100;
   1:  PR[GP1:91,1] = PR[GP1:90,1] + 6.876;
   1:  PR[GP1:91,2] = PR[GP1:90,2] + 9.252;
   1:L PR[91] R[100]mm/sec CNT100;
   1:  PR[GP1:91,1] = PR[GP1:90,1] + 6.205;
   1:  PR[GP1:91,2] = PR[GP1:90,2] + 7.828;
   1:L PR[91] R[100]mm/sec CNT100;
   1:  PR[GP1:91,1] = PR[GP1:90,1] + 5.229;
   1:  PR[GP1:91,2] = PR[GP1:90,2] + 5.609;
   1:L PR[91] R[100]mm/sec CNT100;
   1:  PR[GP1:91,1] = PR[GP1:90,1] + 4.984;
   1:  PR[GP1:91,2] = PR[GP1:90,2] + 4.746;
   1:L PR[91] R[100]mm/sec CNT100;
   1:  PR[GP1:91,1] = PR[GP1:90,1] + 5.031;
   1:  PR[GP1:91,2] = PR[GP1:90,2] + 4.681;
   1:L PR[91] R[100]mm/sec CNT100;
   1:  PR[GP1:91,1] = PR[GP1:90,1] + 4.541;
   1:  PR[GP1:91,2] = PR[GP1:90,2] + 3.314;
   1:L PR[91] R[100]mm/sec CNT100;
   1:  PR[GP1:91,1] = PR[GP1:90,1] + 4.280;
   1:  PR[GP1:91,2] = PR[GP1:90,2] + 3.031;
   1:L PR[91] R[100]mm/sec CNT100;
   1:  PR[GP1:91,1] = PR[GP1:90,1] + 3.799;
   1:  PR[GP1:91,2] = PR[GP1:90,2] + 2.388;
   1:L PR[91] R[100]mm/sec CNT100;
   1:  PR[GP1:91,1] = PR[GP1:90,1] + 3.506;
   1:  PR[GP1:91,2] = PR[GP1:90,2] + 2.184;
   1:L PR[91] R[100]mm/sec CNT100;
   1:  PR[GP1:91,1] = PR[GP1:90,1] + 2.808;
   1:  PR[GP1:91,2] = PR[GP1:90,2] + 1.741;
   1:L PR[91] R[100]mm/sec CNT100;
   1:  PR[GP1:91,1] = PR[GP1:90,1] + 1.814;
   1:  PR[GP1:91,2] = PR[GP1:90,2] + 1.547;
   1:L PR[91] R[100]mm/sec CNT100;
   1:  PR[GP1:91,1] = PR[GP1:90,1] + -1.664;
   1:L PR[91] R[100]mm/sec CNT100;
   1:  PR[91] = PR[90];
   1:  PR[GP1:91,1] = PR[GP1:90,1] + -2.655;
   1:  PR[GP1:91,2] = PR[GP1:90,2] + 2.034;
   1:  PR[GP1:91,3] = PR[GP1:90,3] + 7.625;
   1:L PR[91] R[100]mm/sec CNT100;
   1:  PR[GP1:91,1] = PR[GP1:90,1] + -3.628;
   1:  PR[GP1:91,2] = PR[GP1:90,2] + 2.664;
   1:L PR[91] R[100]mm/sec CNT100;
   1:  PR[GP1:91,1] = PR[GP1:90,1] + -4.138;
   1:  PR[GP1:91,2] = PR[GP1:90,2] + 3.352;
   1:L PR[91] R[100]mm/sec CNT100;
   1:  PR[GP1:91,1] = PR[GP1:90,1] + -4.465;
   1:  PR[GP1:91,2] = PR[GP1:90,2] + 3.733;
   1:L PR[91] R[100]mm/sec CNT100;
   1:  PR[GP1:91,1] = PR[GP1:90,1] + -4.654;
   1:  PR[GP1:91,2] = PR[GP1:90,2] + 4.258;
   1:L PR[91] R[100]mm/sec CNT100;
   1:  PR[GP1:91,1] = PR[GP1:90,1] + -4.905;
   1:  PR[GP1:91,2] = PR[GP1:90,2] + 5.170;
   1:L PR[91] R[100]mm/sec CNT100;
   1:  PR[GP1:91,1] = PR[GP1:90,1] + -5.293;
   1:  PR[GP1:91,2] = PR[GP1:90,2] + 5.992;
   1:L PR[91] R[100]mm/sec CNT100;
   1:  PR[GP1:91,1] = PR[GP1:90,1] + -6.720;
   1:  PR[GP1:91,2] = PR[GP1:90,2] + 9.327;
   1:L PR[91] R[100]mm/sec CNT100;
   1:  PR[GP1:91,1] = PR[GP1:90,1] + -7.315;
   1:  PR[GP1:91,2] = PR[GP1:90,2] + 10.188;
   1:L PR[91] R[100]mm/sec CNT100;
   1:  PR[GP1:91,1] = PR[GP1:90,1] + -9.258;
   1:  PR[GP1:91,2] = PR[GP1:90,2] + 12.639;
   1:L PR[91] R[100]mm/sec CNT100;
   1:  PR[GP1:91,1] = PR[GP1:90,1] + -10.059;
   1:  PR[GP1:91,2] = PR[GP1:90,2] + 13.468;
   1:L PR[91] R[100]mm/sec CNT100;
   1:  PR[GP1:91,1] = PR[GP1:90,1] + -13.449;
   1:  PR[GP1:91,2] = PR[GP1:90,2] + 15.987;
   1:L PR[91] R[100]mm/sec CNT100;
   1:  PR[GP1:91,1] = PR[GP1:90,1] + -14.582;
   1:  PR[GP1:91,2] = PR[GP1:90,2] + 16.570;
   1:L PR[91] R[100]mm/sec CNT100;
   1:  PR[GP1:91,1] = PR[GP1:90,1] + -17.127;
   1:  PR[GP1:91,2] = PR[GP1:90,2] + 17.588;
   1:L PR[91] R[100]mm/sec CNT100;
   1:  PR[GP1:91,1] = PR[GP1:90,1] + -18.473;
   1:  PR[GP1:91,2] = PR[GP1:90,2] + 18.021;
   1:L PR[91] R[100]mm/sec CNT100;
   1:  PR[GP1:91,1] = PR[GP1:90,1] + -19.900;
   1:  PR[GP1:91,2] = PR[GP1:90,2] + 18.234;
   1:L PR[91] R[100]mm/sec CNT100;
   1:  PR[GP1:91,1] = PR[GP1:90,1] + -22.483;
   1:  PR[GP1:91,2] = PR[GP1:90,2] + 18.546;
   1:L PR[91] R[100]mm/sec CNT100;
   1:  PR[GP1:91,1] = PR[GP1:90,1] + -23.960;
   1:  PR[GP1:91,2] = PR[GP1:90,2] + 18.523;
   1:L PR[91] R[100]mm/sec CNT100;
   1:  PR[GP1:91,1] = PR[GP1:90,1] + -25.538;
   1:  PR[GP1:91,2] = PR[GP1:90,2] + 18.237;
   1:L PR[91] R[100]mm/sec CNT100;
   1:  PR[GP1:91,1] = PR[GP1:90,1] + -27.982;
   1:  PR[GP1:91,2] = PR[GP1:90,2] + 17.891;
   1:L PR[91] R[100]mm/sec CNT100;
   1:  PR[GP1:91,1] = PR[GP1:90,1] + -29.495;
   1:  PR[GP1:91,2] = PR[GP1:90,2] + 17.351;
   1:L PR[91] R[100]mm/sec CNT100;
   1:  PR[GP1:91,1] = PR[GP1:90,1] + -31.579;
   1:  PR[GP1:91,2] = PR[GP1:90,2] + 16.473;
   1:L PR[91] R[100]mm/sec CNT100;
   1:  PR[GP1:91,1] = PR[GP1:90,1] + -33.047;
   1:  PR[GP1:91,2] = PR[GP1:90,2] + 15.659;
   1:L PR[91] R[100]mm/sec CNT100;
   1:  PR[GP1:91,1] = PR[GP1:90,1] + -34.429;
   1:  PR[GP1:91,2] = PR[GP1:90,2] + 14.562;
   1:L PR[91] R[100]mm/sec CNT100;
   1:  PR[GP1:91,1] = PR[GP1:90,1] + -36.143;
   1:  PR[GP1:91,2] = PR[GP1:90,2] + 13.235;
   1:L PR[91] R[100]mm/sec CNT100;
   1:  PR[GP1:91,1] = PR[GP1:90,1] + -37.318;
   1:  PR[GP1:91,2] = PR[GP1:90,2] + 11.939;
   1:L PR[91] R[100]mm/sec CNT100;
   1:  PR[GP1:91,1] = PR[GP1:90,1] + -38.558;
   1:  PR[GP1:91,2] = PR[GP1:90,2] + 10.313;
   1:L PR[91] R[100]mm/sec CNT100;
   1:  PR[GP1:91,1] = PR[GP1:90,1] + -39.538;
   1:  PR[GP1:91,2] = PR[GP1:90,2] + 8.794;
   1:L PR[91] R[100]mm/sec CNT100;
   1:  PR[GP1:91,1] = PR[GP1:90,1] + -40.275;
   1:  PR[GP1:91,2] = PR[GP1:90,2] + 7.096;
   1:L PR[91] R[100]mm/sec CNT100;
   1:  PR[GP1:91,1] = PR[GP1:90,1] + -41.036;
   1:  PR[GP1:91,2] = PR[GP1:90,2] + 5.253;
   1:L PR[91] R[100]mm/sec CNT100;
   1:  PR[GP1:91,1] = PR[GP1:90,1] + -41.470;
   1:  PR[GP1:91,2] = PR[GP1:90,2] + 3.521;
   1:L PR[91] R[100]mm/sec CNT100;
   1:  PR[GP1:91,1] = PR[GP1:90,1] + -41.627;
   1:  PR[GP1:91,2] = PR[GP1:90,2] + 1.603;
   1:L PR[91] R[100]mm/sec CNT100;
   1:  PR[GP1:91,1] = PR[GP1:90,1] + -41.880;
   1:  PR[GP1:91,2] = PR[GP1:90,2] + -0.346;
   1:L PR[91] R[100]mm/sec CNT100;
   1:  PR[GP1:91,1] = PR[GP1:90,1] + -41.728;
   1:  PR[GP1:91,2] = PR[GP1:90,2] + -2.203;
   1:L PR[91] R[100]mm/sec CNT100;
   1:  PR[GP1:91,1] = PR[GP1:90,1] + -41.478;
   1:  PR[GP1:91,2] = PR[GP1:90,2] + -4.112;
   1:L PR[91] R[100]mm/sec CNT100;
   1:  PR[GP1:91,1] = PR[GP1:90,1] + -41.039;
   1:  PR[GP1:91,2] = PR[GP1:90,2] + -5.865;
   1:L PR[91] R[100]mm/sec CNT100;
   1:  PR[GP1:91,1] = PR[GP1:90,1] + -40.282;
   1:  PR[GP1:91,2] = PR[GP1:90,2] + -7.611;
   1:L PR[91] R[100]mm/sec CNT100;
   1:  PR[GP1:91,1] = PR[GP1:90,1] + -39.531;
   1:  PR[GP1:91,2] = PR[GP1:90,2] + -9.429;
   1:L PR[91] R[100]mm/sec CNT100;
   1:  PR[GP1:91,1] = PR[GP1:90,1] + -38.558;
   1:  PR[GP1:91,2] = PR[GP1:90,2] + -10.937;
   1:L PR[91] R[100]mm/sec CNT100;
   1:  PR[GP1:91,1] = PR[GP1:90,1] + -37.318;
   1:  PR[GP1:91,2] = PR[GP1:90,2] + -12.563;
   1:L PR[91] R[100]mm/sec CNT100;
   1:  PR[GP1:91,1] = PR[GP1:90,1] + -36.137;
   1:  PR[GP1:91,2] = PR[GP1:90,2] + -13.865;
   1:L PR[91] R[100]mm/sec CNT100;
   1:  PR[GP1:91,1] = PR[GP1:90,1] + -34.718;
   1:  PR[GP1:91,2] = PR[GP1:90,2] + -14.991;
   1:L PR[91] R[100]mm/sec CNT100;
   1:  PR[GP1:91,1] = PR[GP1:90,1] + -33.054;
   1:  PR[GP1:91,2] = PR[GP1:90,2] + -16.278;
   1:L PR[91] R[100]mm/sec CNT100;
   1:  PR[GP1:91,1] = PR[GP1:90,1] + -31.580;
   1:  PR[GP1:91,2] = PR[GP1:90,2] + -17.097;
   1:L PR[91] R[100]mm/sec CNT100;
   1:  PR[GP1:91,1] = PR[GP1:90,1] + -29.495;
   1:  PR[GP1:91,2] = PR[GP1:90,2] + -17.975;
   1:L PR[91] R[100]mm/sec CNT100;
   1:  PR[GP1:91,1] = PR[GP1:90,1] + -27.955;
   1:  PR[GP1:91,2] = PR[GP1:90,2] + -18.525;
   1:L PR[91] R[100]mm/sec CNT100;
   1:  PR[GP1:91,1] = PR[GP1:90,1] + -26.336;
   1:  PR[GP1:91,2] = PR[GP1:90,2] + -18.819;
   1:L PR[91] R[100]mm/sec CNT100;
   1:  PR[GP1:91,1] = PR[GP1:90,1] + -23.990;
   1:  PR[GP1:91,2] = PR[GP1:90,2] + -19.147;
   1:L PR[91] R[100]mm/sec CNT100;
   1:  PR[GP1:91,1] = PR[GP1:90,1] + -22.503;
   1:  PR[GP1:91,2] = PR[GP1:90,2] + -19.170;
   1:L PR[91] R[100]mm/sec CNT100;
   1:  PR[GP1:91,1] = PR[GP1:90,1] + -20.924;
   1:  PR[GP1:91,2] = PR[GP1:90,2] + -18.935;
   1:L PR[91] R[100]mm/sec CNT100;
   1:  PR[GP1:91,1] = PR[GP1:90,1] + -18.453;
   1:  PR[GP1:91,2] = PR[GP1:90,2] + -18.639;
   1:L PR[91] R[100]mm/sec CNT100;
   1:  PR[GP1:91,1] = PR[GP1:90,1] + -17.128;
   1:  PR[GP1:91,2] = PR[GP1:90,2] + -18.212;
   1:L PR[91] R[100]mm/sec CNT100;
   1:  PR[GP1:91,1] = PR[GP1:90,1] + -14.582;
   1:  PR[GP1:91,2] = PR[GP1:90,2] + -17.194;
   1:L PR[91] R[100]mm/sec CNT100;
   1:  PR[GP1:91,1] = PR[GP1:90,1] + -13.450;
   1:  PR[GP1:91,2] = PR[GP1:90,2] + -16.612;
   1:L PR[91] R[100]mm/sec CNT100;
   1:  PR[GP1:91,1] = PR[GP1:90,1] + -10.059;
   1:  PR[GP1:91,2] = PR[GP1:90,2] + -14.092;
   1:L PR[91] R[100]mm/sec CNT100;
   1:  PR[GP1:91,1] = PR[GP1:90,1] + -9.258;
   1:  PR[GP1:91,2] = PR[GP1:90,2] + -13.263;
   1:L PR[91] R[100]mm/sec CNT100;
   1:  PR[GP1:91,1] = PR[GP1:90,1] + -7.315;
   1:  PR[GP1:91,2] = PR[GP1:90,2] + -10.813;
   1:L PR[91] R[100]mm/sec CNT100;
   1:  PR[GP1:91,1] = PR[GP1:90,1] + -6.705;
   1:  PR[GP1:91,2] = PR[GP1:90,2] + -9.930;
   1:L PR[91] R[100]mm/sec CNT100;
   1:  PR[GP1:91,1] = PR[GP1:90,1] + -6.237;
   1:  PR[GP1:91,2] = PR[GP1:90,2] + -8.937;
   1:L PR[91] R[100]mm/sec CNT100;
   1:  PR[GP1:91,1] = PR[GP1:90,1] + -4.946;
   1:  PR[GP1:91,2] = PR[GP1:90,2] + -5.970;
   1:L PR[91] R[100]mm/sec CNT100;
   1:  PR[GP1:91,1] = PR[GP1:90,1] + -4.647;
   1:  PR[GP1:91,2] = PR[GP1:90,2] + -4.884;
   1:L PR[91] R[100]mm/sec CNT100;
   1:  PR[GP1:91,1] = PR[GP1:90,1] + -4.440;
   1:  PR[GP1:91,2] = PR[GP1:90,2] + -4.310;
   1:L PR[91] R[100]mm/sec CNT100;
   1:  PR[GP1:91,1] = PR[GP1:90,1] + -4.127;
   1:  PR[GP1:91,2] = PR[GP1:90,2] + -3.962;
   1:L PR[91] R[100]mm/sec CNT100;
   1:  PR[GP1:91,1] = PR[GP1:90,1] + -3.627;
   1:  PR[GP1:91,2] = PR[GP1:90,2] + -3.288;
   1:L PR[91] R[100]mm/sec CNT100;
   1:  PR[GP1:91,1] = PR[GP1:90,1] + -2.655;
   1:  PR[GP1:91,2] = PR[GP1:90,2] + -2.658;
   1:L PR[91] R[100]mm/sec CNT100;
   1:  PR[GP1:91,1] = PR[GP1:90,1] + -1.655;
   1:  PR[GP1:91,2] = PR[GP1:90,2] + -2.459;
   1:L PR[91] R[100]mm/sec CNT100;
   1:  PR[GP1:91,1] = PR[GP1:90,1] + 1.808;
   1:L PR[91] R[100]mm/sec CNT100;
   1:  PR[GP1:91,1] = PR[GP1:90,1] + 2.810;
   1:  PR[GP1:91,2] = PR[GP1:90,2] + -2.657;
   1:L PR[91] R[100]mm/sec CNT100;
   1:  PR[GP1:91,1] = PR[GP1:90,1] + 3.783;
   1:  PR[GP1:91,2] = PR[GP1:90,2] + -3.287;
   1:L PR[91] R[100]mm/sec CNT100;
   1:  PR[GP1:91,1] = PR[GP1:90,1] + 4.291;
   1:  PR[GP1:91,2] = PR[GP1:90,2] + -3.973;
   1:L PR[91] R[100]mm/sec CNT100;
   1:  PR[GP1:91,1] = PR[GP1:90,1] + 4.616;
   1:  PR[GP1:91,2] = PR[GP1:90,2] + -4.348;
   1:L PR[91] R[100]mm/sec CNT100;
   1:  PR[GP1:91,1] = PR[GP1:90,1] + 4.809;
   1:  PR[GP1:91,2] = PR[GP1:90,2] + -4.883;
   1:L PR[91] R[100]mm/sec CNT100;
   1:  PR[GP1:91,1] = PR[GP1:90,1] + 5.069;
   1:  PR[GP1:91,2] = PR[GP1:90,2] + -5.824;
   1:L PR[91] R[100]mm/sec CNT100;
   1:  PR[GP1:91,1] = PR[GP1:90,1] + 5.469;
   1:  PR[GP1:91,2] = PR[GP1:90,2] + -6.674;
   1:L PR[91] R[100]mm/sec CNT100;
   1:  PR[GP1:91,1] = PR[GP1:90,1] + 6.876;
   1:  PR[GP1:91,2] = PR[GP1:90,2] + -9.949;
   1:L PR[91] R[100]mm/sec CNT100;
   1:  PR[GP1:91,1] = PR[GP1:90,1] + 7.471;
   1:  PR[GP1:91,2] = PR[GP1:90,2] + -10.810;
   1:L PR[91] R[100]mm/sec CNT100;
   1:  PR[GP1:91,1] = PR[GP1:90,1] + 9.414;
   1:  PR[GP1:91,2] = PR[GP1:90,2] + -13.263;
   1:L PR[91] R[100]mm/sec CNT100;
   1:  PR[GP1:91,1] = PR[GP1:90,1] + 10.215;
   1:  PR[GP1:91,2] = PR[GP1:90,2] + -14.092;
   1:L PR[91] R[100]mm/sec CNT100;
   1:  PR[GP1:91,1] = PR[GP1:90,1] + 13.606;
   1:  PR[GP1:91,2] = PR[GP1:90,2] + -16.611;
   1:L PR[91] R[100]mm/sec CNT100;
   1:  PR[GP1:91,1] = PR[GP1:90,1] + 14.738;
   1:  PR[GP1:91,2] = PR[GP1:90,2] + -17.194;
   1:L PR[91] R[100]mm/sec CNT100;
   1:  PR[GP1:91,1] = PR[GP1:90,1] + 17.284;
   1:  PR[GP1:91,2] = PR[GP1:90,2] + -18.212;
   1:L PR[91] R[100]mm/sec CNT100;
   1:  PR[GP1:91,1] = PR[GP1:90,1] + 18.629;
   1:  PR[GP1:91,2] = PR[GP1:90,2] + -18.645;
   1:L PR[91] R[100]mm/sec CNT100;
   1:  PR[GP1:91,1] = PR[GP1:90,1] + 20.056;
   1:  PR[GP1:91,2] = PR[GP1:90,2] + -18.858;
   1:L PR[91] R[100]mm/sec CNT100;
   1:  PR[GP1:91,1] = PR[GP1:90,1] + 22.639;
   1:  PR[GP1:91,2] = PR[GP1:90,2] + -19.171;
   1:L PR[91] R[100]mm/sec CNT100;
   1:  PR[GP1:91,1] = PR[GP1:90,1] + 24.117;
   1:  PR[GP1:91,2] = PR[GP1:90,2] + -19.147;
   1:L PR[91] R[100]mm/sec CNT100;
   1:  PR[GP1:91,1] = PR[GP1:90,1] + 25.695;
   1:  PR[GP1:91,2] = PR[GP1:90,2] + -18.861;
   1:L PR[91] R[100]mm/sec CNT100;
   1:  PR[GP1:91,1] = PR[GP1:90,1] + 28.138;
   1:  PR[GP1:91,2] = PR[GP1:90,2] + -18.515;
   1:L PR[91] R[100]mm/sec CNT100;
   1:  PR[GP1:91,1] = PR[GP1:90,1] + 29.651;
   1:  PR[GP1:91,2] = PR[GP1:90,2] + -17.975;
   1:L PR[91] R[100]mm/sec CNT100;
   1:  PR[GP1:91,1] = PR[GP1:90,1] + 31.736;
   1:  PR[GP1:91,2] = PR[GP1:90,2] + -17.097;
   1:L PR[91] R[100]mm/sec CNT100;
   1:  PR[GP1:91,1] = PR[GP1:90,1] + 33.203;
   1:  PR[GP1:91,2] = PR[GP1:90,2] + -16.283;
   1:L PR[91] R[100]mm/sec CNT100;
   1:  PR[GP1:91,1] = PR[GP1:90,1] + 34.586;
   1:  PR[GP1:91,2] = PR[GP1:90,2] + -15.186;
   1:L PR[91] R[100]mm/sec CNT100;
   1:  PR[GP1:91,1] = PR[GP1:90,1] + 36.299;
   1:  PR[GP1:91,2] = PR[GP1:90,2] + -13.859;
   1:L PR[91] R[100]mm/sec CNT100;
   1:  PR[GP1:91,1] = PR[GP1:90,1] + 37.475;
   1:  PR[GP1:91,2] = PR[GP1:90,2] + -12.563;
   1:L PR[91] R[100]mm/sec CNT100;
   1:  PR[GP1:91,1] = PR[GP1:90,1] + 38.715;
   1:  PR[GP1:91,2] = PR[GP1:90,2] + -10.937;
   1:L PR[91] R[100]mm/sec CNT100;
   1:  PR[GP1:91,1] = PR[GP1:90,1] + 39.695;
   1:  PR[GP1:91,2] = PR[GP1:90,2] + -9.418;
   1:L PR[91] R[100]mm/sec CNT100;
   1:  PR[GP1:91,1] = PR[GP1:90,1] + 40.431;
   1:  PR[GP1:91,2] = PR[GP1:90,2] + -7.719;
   1:L PR[91] R[100]mm/sec CNT100;
   1:  PR[GP1:91,1] = PR[GP1:90,1] + 41.193;
   1:  PR[GP1:91,2] = PR[GP1:90,2] + -5.878;
   1:L PR[91] R[100]mm/sec CNT100;
   1:  PR[GP1:91,1] = PR[GP1:90,1] + 41.627;
   1:  PR[GP1:91,2] = PR[GP1:90,2] + -4.147;
   1:L PR[91] R[100]mm/sec CNT100;
   1:  PR[GP1:91,1] = PR[GP1:90,1] + 41.784;
   1:  PR[GP1:91,2] = PR[GP1:90,2] + -2.229;
   1:L PR[91] R[100]mm/sec CNT100;
   1:  PR[GP1:91,1] = PR[GP1:90,1] + 42.037;
   1:  PR[GP1:91,2] = PR[GP1:90,2] + -0.278;
   1:L PR[91] R[100]mm/sec CNT100;
   1:  PR[GP1:91,1] = PR[GP1:90,1] + 41.885;
   1:  PR[GP1:91,2] = PR[GP1:90,2] + 1.579;
   1:L PR[91] R[100]mm/sec CNT100;
   1:  PR[GP1:91,1] = PR[GP1:90,1] + 41.635;
   1:  PR[GP1:91,2] = PR[GP1:90,2] + 3.490;
   1:L PR[91] R[100]mm/sec CNT100;
   1:  PR[GP1:91,1] = PR[GP1:90,1] + 41.196;
   1:  PR[GP1:91,2] = PR[GP1:90,2] + 5.243;
   1:L PR[91] R[100]mm/sec CNT100;
   1:  PR[GP1:91,1] = PR[GP1:90,1] + 40.438;
   1:  PR[GP1:91,2] = PR[GP1:90,2] + 6.989;
   1:L PR[91] R[100]mm/sec CNT100;
   1:  PR[GP1:91,1] = PR[GP1:90,1] + 39.687;
   1:  PR[GP1:91,2] = PR[GP1:90,2] + 8.805;
   1:L PR[91] R[100]mm/sec CNT100;
   1:  PR[GP1:91,1] = PR[GP1:90,1] + 38.714;
   1:  PR[GP1:91,2] = PR[GP1:90,2] + 10.314;
   1:L PR[91] R[100]mm/sec CNT100;
   1:  PR[GP1:91,1] = PR[GP1:90,1] + 37.474;
   1:  PR[GP1:91,2] = PR[GP1:90,2] + 11.940;
   1:L PR[91] R[100]mm/sec CNT100;
   1:  PR[GP1:91,1] = PR[GP1:90,1] + 36.293;
   1:  PR[GP1:91,2] = PR[GP1:90,2] + 13.242;
   1:L PR[91] R[100]mm/sec CNT100;
   1:  PR[GP1:91,1] = PR[GP1:90,1] + 34.874;
   1:  PR[GP1:91,2] = PR[GP1:90,2] + 14.368;
   1:L PR[91] R[100]mm/sec CNT100;
   1:  PR[GP1:91,1] = PR[GP1:90,1] + 33.209;
   1:  PR[GP1:91,2] = PR[GP1:90,2] + 15.656;
   1:L PR[91] R[100]mm/sec CNT100;
   1:  PR[GP1:91,1] = PR[GP1:90,1] + 31.734;
   1:  PR[GP1:91,2] = PR[GP1:90,2] + 16.474;
   1:L PR[91] R[100]mm/sec CNT100;
   1:  PR[GP1:91,1] = PR[GP1:90,1] + 29.649;
   1:  PR[GP1:91,2] = PR[GP1:90,2] + 17.352;
   1:L PR[91] R[100]mm/sec CNT100;
   1:  PR[GP1:91,1] = PR[GP1:90,1] + 28.109;
   1:  PR[GP1:91,2] = PR[GP1:90,2] + 17.902;
   1:L PR[91] R[100]mm/sec CNT100;
   1:  PR[GP1:91,1] = PR[GP1:90,1] + 26.490;
   1:  PR[GP1:91,2] = PR[GP1:90,2] + 18.195;
   1:L PR[91] R[100]mm/sec CNT100;
   1:  PR[GP1:91,1] = PR[GP1:90,1] + 24.143;
   1:  PR[GP1:91,2] = PR[GP1:90,2] + 18.523;
   1:L PR[91] R[100]mm/sec CNT100;
   1:  PR[GP1:91,1] = PR[GP1:90,1] + 22.656;
   1:  PR[GP1:91,2] = PR[GP1:90,2] + 18.546;
   1:L PR[91] R[100]mm/sec CNT100;
   1:  PR[GP1:91,1] = PR[GP1:90,1] + 21.077;
   1:  PR[GP1:91,2] = PR[GP1:90,2] + 18.311;
   1:L PR[91] R[100]mm/sec CNT100;
   1:  PR[GP1:91,1] = PR[GP1:90,1] + 18.605;
   1:  PR[GP1:91,2] = PR[GP1:90,2] + 18.014;
   1:L PR[91] R[100]mm/sec CNT100;
   1:  PR[GP1:91,1] = PR[GP1:90,1] + 17.280;
   1:  PR[GP1:91,2] = PR[GP1:90,2] + 17.587;
   1:L PR[91] R[100]mm/sec CNT100;
   1:  PR[GP1:91,1] = PR[GP1:90,1] + 14.733;
   1:  PR[GP1:91,2] = PR[GP1:90,2] + 16.567;
   1:L PR[91] R[100]mm/sec CNT100;
   1:  PR[GP1:91,1] = PR[GP1:90,1] + 13.601;
   1:  PR[GP1:91,2] = PR[GP1:90,2] + 15.985;
   1:L PR[91] R[100]mm/sec CNT100;
   1:  PR[GP1:91,1] = PR[GP1:90,1] + 10.211;
   1:  PR[GP1:91,2] = PR[GP1:90,2] + 13.463;
   1:L PR[91] R[100]mm/sec CNT100;
   1:  PR[GP1:91,1] = PR[GP1:90,1] + 9.410;
   1:  PR[GP1:91,2] = PR[GP1:90,2] + 12.635;
   1:L PR[91] R[100]mm/sec CNT100;
   1:  PR[GP1:91,1] = PR[GP1:90,1] + 7.467;
   1:  PR[GP1:91,2] = PR[GP1:90,2] + 10.180;
   1:L PR[91] R[100]mm/sec CNT100;
   1:  PR[GP1:91,1] = PR[GP1:90,1] + 6.858;
   1:  PR[GP1:91,2] = PR[GP1:90,2] + 9.297;
   1:L PR[91] R[100]mm/sec CNT100;
   1:  PR[GP1:91,1] = PR[GP1:90,1] + 6.388;
   1:  PR[GP1:91,2] = PR[GP1:90,2] + 8.301;
   1:L PR[91] R[100]mm/sec CNT100;
   1:  PR[GP1:91,1] = PR[GP1:90,1] + 5.112;
   1:  PR[GP1:91,2] = PR[GP1:90,2] + 5.397;
   1:L PR[91] R[100]mm/sec CNT100;
   1:  PR[GP1:91,1] = PR[GP1:90,1] + 4.996;
   1:  PR[GP1:91,2] = PR[GP1:90,2] + 4.991;
   1:L PR[91] R[100]mm/sec CNT100;
   1:  PR[GP1:91,1] = PR[GP1:90,1] + 5.040;
   1:  PR[GP1:91,2] = PR[GP1:90,2] + 4.931;
   1:L PR[91] R[100]mm/sec CNT100;
   1:  PR[GP1:91,1] = PR[GP1:90,1] + 4.610;
   1:  PR[GP1:91,2] = PR[GP1:90,2] + 3.731;
   1:L PR[91] R[100]mm/sec CNT100;
   1:  PR[GP1:91,1] = PR[GP1:90,1] + 4.294;
   1:  PR[GP1:91,2] = PR[GP1:90,2] + 3.318;
   1:L PR[91] R[100]mm/sec CNT100;
   1:  PR[GP1:91,1] = PR[GP1:90,1] + 4.224;
   1:  PR[GP1:91,2] = PR[GP1:90,2] + 3.259;
   1:L PR[91] R[100]mm/sec CNT100;
   1:  PR[GP1:91,1] = PR[GP1:90,1] + 3.799;
   1:  PR[GP1:91,2] = PR[GP1:90,2] + 2.684;
   1:L PR[91] R[100]mm/sec CNT100;
   1:  PR[GP1:91,1] = PR[GP1:90,1] + 3.461;
   1:  PR[GP1:91,2] = PR[GP1:90,2] + 2.449;
   1:L PR[91] R[100]mm/sec CNT100;
   1:  PR[GP1:91,1] = PR[GP1:90,1] + 2.803;
   1:  PR[GP1:91,2] = PR[GP1:90,2] + 2.032;
   1:L PR[91] R[100]mm/sec CNT100;
   1:  PR[GP1:91,1] = PR[GP1:90,1] + 1.806;
   1:  PR[GP1:91,2] = PR[GP1:90,2] + 1.835;
   1:L PR[91] R[100]mm/sec CNT100;
   1:  PR[GP1:91,1] = PR[GP1:90,1] + -1.660;
   1:L PR[91] R[100]mm/sec CNT100;
   1:  PR[91] = PR[90];
   1:  PR[GP1:91,1] = PR[GP1:90,1] + -2.654;
   1:  PR[GP1:91,2] = PR[GP1:90,2] + 2.326;
   1:  PR[GP1:91,3] = PR[GP1:90,3] + 8.235;
   1:L PR[91] R[100]mm/sec CNT100;
   1:  PR[GP1:91,1] = PR[GP1:90,1] + -3.629;
   1:  PR[GP1:91,2] = PR[GP1:90,2] + 2.962;
   1:L PR[91] R[100]mm/sec CNT100;
   1:  PR[GP1:91,1] = PR[GP1:90,1] + -4.136;
   1:  PR[GP1:91,2] = PR[GP1:90,2] + 3.654;
   1:L PR[91] R[100]mm/sec CNT100;
   1:  PR[GP1:91,1] = PR[GP1:90,1] + -4.550;
   1:  PR[GP1:91,2] = PR[GP1:90,2] + 4.136;
   1:L PR[91] R[100]mm/sec CNT100;
   1:  PR[GP1:91,1] = PR[GP1:90,1] + -4.772;
   1:  PR[GP1:91,2] = PR[GP1:90,2] + 4.899;
   1:L PR[91] R[100]mm/sec CNT100;
   1:  PR[GP1:91,1] = PR[GP1:90,1] + -4.940;
   1:  PR[GP1:91,2] = PR[GP1:90,2] + 5.255;
   1:L PR[91] R[100]mm/sec CNT100;
   1:  PR[GP1:91,1] = PR[GP1:90,1] + -6.702;
   1:  PR[GP1:91,2] = PR[GP1:90,2] + 9.374;
   1:L PR[91] R[100]mm/sec CNT100;
   1:  PR[GP1:91,1] = PR[GP1:90,1] + -7.028;
   1:  PR[GP1:91,2] = PR[GP1:90,2] + 9.845;
   1:L PR[91] R[100]mm/sec CNT100;
   1:  PR[GP1:91,1] = PR[GP1:90,1] + -9.430;
   1:  PR[GP1:91,2] = PR[GP1:90,2] + 12.875;
   1:L PR[91] R[100]mm/sec CNT100;
   1:  PR[GP1:91,1] = PR[GP1:90,1] + -9.918;
   1:  PR[GP1:91,2] = PR[GP1:90,2] + 13.380;
   1:L PR[91] R[100]mm/sec CNT100;
   1:  PR[GP1:91,1] = PR[GP1:90,1] + -13.517;
   1:  PR[GP1:91,2] = PR[GP1:90,2] + 16.055;
   1:L PR[91] R[100]mm/sec CNT100;
   1:  PR[GP1:91,1] = PR[GP1:90,1] + -14.273;
   1:  PR[GP1:91,2] = PR[GP1:90,2] + 16.444;
   1:L PR[91] R[100]mm/sec CNT100;
   1:  PR[GP1:91,1] = PR[GP1:90,1] + -17.423;
   1:  PR[GP1:91,2] = PR[GP1:90,2] + 17.703;
   1:L PR[91] R[100]mm/sec CNT100;
   1:  PR[GP1:91,1] = PR[GP1:90,1] + -18.392;
   1:  PR[GP1:91,2] = PR[GP1:90,2] + 18.015;
   1:L PR[91] R[100]mm/sec CNT100;
   1:  PR[GP1:91,1] = PR[GP1:90,1] + -19.428;
   1:  PR[GP1:91,2] = PR[GP1:90,2] + 18.170;
   1:L PR[91] R[100]mm/sec CNT100;
   1:  PR[GP1:91,1] = PR[GP1:90,1] + -22.626;
   1:  PR[GP1:91,2] = PR[GP1:90,2] + 18.557;
   1:L PR[91] R[100]mm/sec CNT100;
   1:  PR[GP1:91,1] = PR[GP1:90,1] + -23.733;
   1:  PR[GP1:91,2] = PR[GP1:90,2] + 18.539;
   1:L PR[91] R[100]mm/sec CNT100;
   1:  PR[GP1:91,1] = PR[GP1:90,1] + -24.947;
   1:  PR[GP1:91,2] = PR[GP1:90,2] + 18.319;
   1:L PR[91] R[100]mm/sec CNT100;
   1:  PR[GP1:91,1] = PR[GP1:90,1] + -27.973;
   1:  PR[GP1:91,2] = PR[GP1:90,2] + 17.891;
   1:L PR[91] R[100]mm/sec CNT100;
   1:  PR[GP1:91,1] = PR[GP1:90,1] + -29.159;
   1:  PR[GP1:91,2] = PR[GP1:90,2] + 17.467;
   1:L PR[91] R[100]mm/sec CNT100;
   1:  PR[GP1:91,1] = PR[GP1:90,1] + -31.743;
   1:  PR[GP1:91,2] = PR[GP1:90,2] + 16.379;
   1:L PR[91] R[100]mm/sec CNT100;
   1:  PR[GP1:91,1] = PR[GP1:90,1] + -32.923;
   1:  PR[GP1:91,2] = PR[GP1:90,2] + 15.724;
   1:L PR[91] R[100]mm/sec CNT100;
   1:  PR[GP1:91,1] = PR[GP1:90,1] + -34.047;
   1:  PR[GP1:91,2] = PR[GP1:90,2] + 14.832;
   1:L PR[91] R[100]mm/sec CNT100;
   1:  PR[GP1:91,1] = PR[GP1:90,1] + -36.172;
   1:  PR[GP1:91,2] = PR[GP1:90,2] + 13.187;
   1:L PR[91] R[100]mm/sec CNT100;
   1:  PR[GP1:91,1] = PR[GP1:90,1] + -37.137;
   1:  PR[GP1:91,2] = PR[GP1:90,2] + 12.124;
   1:L PR[91] R[100]mm/sec CNT100;
   1:  PR[GP1:91,1] = PR[GP1:90,1] + -38.675;
   1:  PR[GP1:91,2] = PR[GP1:90,2] + 10.106;
   1:L PR[91] R[100]mm/sec CNT100;
   1:  PR[GP1:91,1] = PR[GP1:90,1] + -39.490;
   1:  PR[GP1:91,2] = PR[GP1:90,2] + 8.843;
   1:L PR[91] R[100]mm/sec CNT100;
   1:  PR[GP1:91,1] = PR[GP1:90,1] + -40.106;
   1:  PR[GP1:91,2] = PR[GP1:90,2] + 7.424;
   1:L PR[91] R[100]mm/sec CNT100;
